KUKA KRL program: EPS_2_25694_LG03_A_20260223033042.src

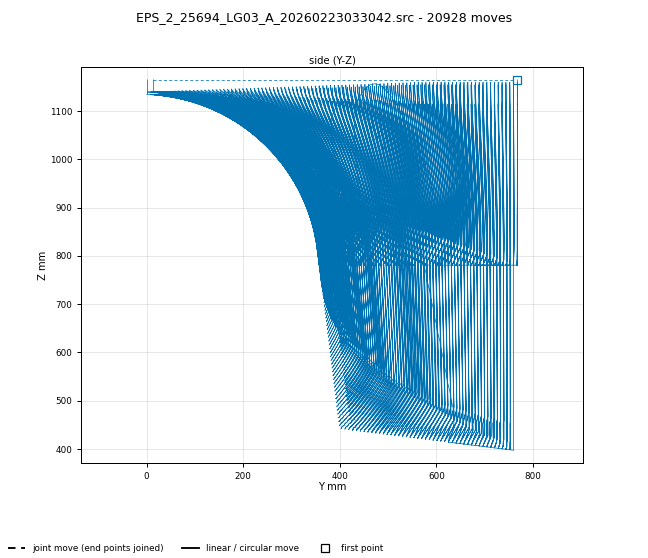
[picture p0: tool path of EPS_2_25694_LG03_A_20260223033042.src, 20928 of 20930 moves have a stored position in this frame; points joined in program order, loops and branches not executed]
&ACCESS RVP
&REL 4
&COMMENT QRS 19112012
&PARAM EDITMASK = *
DEF PART()
EXT BAS (BAS_COMMAND :IN,REAL :IN )
INT I
BAS (#INITMOV,0 )

;KUKA QRS Post kuka4.cps  Date:22-06-2017 !

File_ID=3046

QRS_PRE_INIT()

;Init var - Until changes are made in qrs_pre_init
Outlet_Square_prg=0
Inlet_1_Square_prg=0
Inlet_2_Square_prg=0
Inlet_3_Square_prg=0
Inlet_4_Square_prg=0
Inlet_5_Square_prg=0

Outlet_1={X 0.000, Y 562.000, Z 811.500, B 0.000, E1 0.000 }
Inlet_1={X 0.000, Y 562.000, Z 771.500, B 0.000, E1 183.000 }
Outlet_1_type=686
Inlet_1_type=686
;QRS#1=Sidecore dimensions
;QRS#2=675-27" Concrete
;QRS#3=675-27" Concrete
;QRS#4=
;QRS#5=
;QRS#6=
;QRS#7=
;QRS#8=
;QRS#9=S306-38L
;QRS#10=S306-38L
;QRS#11=
;QRS#12=
;QRS#13=
;QRS#14=
;QRS#15=
;QRS#16=1524x152x1600 5,25'
;QRS#17=EPS Height
;QRS#18=1154,5
;QRS#19=*
;QRS#20= UPDATED VERSION 22-06-2017
;QRS#21=*
Outlet_Square=0550
Inlet_1_Square=0550
Inlet_2_Square=0
Inlet_3_Square=0
Inlet_4_Square=0
Inlet_5_Square=0
Mill_Square=1
Outlet_Square_Prg=265
Inlet_1_Square_prg=265

QRS_INIT()

$ADVANCE=5

; T1
PTP {E1 173.017,E2 173.017}
PTP {X 0,Y 767.74,A -85,B 0,C 180,E1 173.017,E2 173.017,E3 0,E4 0,E5 0,E6 0}
QRS_SPEED_INIT()
LIN {X 0,Y 767.74,Z 1164.5,A -85,B 0,C 180,E1 173.017,E2 173.017,E3 0,E4 0,E5 0,E6 0} C_VEL
LIN {X 0,Y 767.74,Z 782.81,A -85,B 0,C 180,E1 173.017,E2 173.017} C_VEL
LIN {X 0,Y 767.776,Z 780.81,A -85,B 0,C 180,E1 173.166,E2 173.166} C_VEL
LIN {X 0,Y 767.86,Z 780.81,A -85,B 0,C 180,E1 173.458,E2 173.458} C_VEL
LIN {X 0,Y 767.876,Z 780.81,A -85,B 0,C 180,E1 177.201,E2 177.201} C_VEL
LIN {X 0,Y 767.864,Z 780.81,A -85,B 0,C 180,E1 180.933,E2 180.933} C_VEL
LIN {X 0,Y 767.829,Z 780.81,A -85,B 0,C 180,E1 184.668,E2 184.668} C_VEL
LIN {X 0,Y 767.837,Z 780.81,A -85,B 0,C 180,E1 188.423,E2 188.423} C_VEL
LIN {X 0,Y 767.822,Z 780.81,A -85,B 0,C 180,E1 192.215,E2 192.215} C_VEL
LIN {X 0,Y 767.843,Z 780.81,A -85,B 0,C 180,E1 196.207,E2 196.207} C_VEL
LIN {X 0,Y 767.794,Z 780.81,A -85,B 0,C 180,E1 199.987,E2 199.987} C_VEL
LIN {X 0,Y 767.77,Z 780.81,A -85,B 0,C 180,E1 204.012,E2 204.012} C_VEL
LIN {X 0,Y 767.76,Z 780.81,A -85,B 0,C 180,E1 208.167,E2 208.167} C_VEL
LIN {X 0,Y 767.325,Z 780.81,A -85,B 0,C 180,E1 210.324,E2 210.324} C_VEL
LIN {X 0,Y 767.754,Z 780.81,A -85,B 0,C 180,E1 212.49,E2 212.49} C_VEL
LIN {X 0,Y 767.438,Z 780.81,A -85,B 0,C 180,E1 213.851,E2 213.851} C_VEL
LIN {X 0,Y 767.747,Z 780.81,A -85,B 0,C 180,E1 217.098,E2 217.098} C_VEL
LIN {X 0,Y 767.106,Z 780.81,A -85,B 0,C 180,E1 220.032,E2 220.032} C_VEL
LIN {X 0,Y 767.543,Z 780.81,A -85,B 0,C 180,E1 221.879,E2 221.879} C_VEL
LIN {X 0,Y 767.594,Z 780.81,A -85,B 0,C 180,E1 222.892,E2 222.892} C_VEL
LIN {X 0,Y 767.642,Z 780.81,A -85,B 0,C 180,E1 227.104,E2 227.104} C_VEL
LIN {X 0,Y 767.576,Z 780.81,A -85,B 0,C 180,E1 228.123,E2 228.123} C_VEL
LIN {X 0,Y 767.128,Z 780.81,A -85,B 0,C 180,E1 230.555,E2 230.555} C_VEL
LIN {X 0,Y 767.697,Z 780.81,A -85,B 0,C 180,E1 232.964,E2 232.964} C_VEL
LIN {X 0,Y 767.564,Z 780.81,A -85,B 0,C 180,E1 236.135,E2 236.135} C_VEL
LIN {X 0,Y 767.581,Z 780.81,A -85,B 0,C 180,E1 237.502,E2 237.502} C_VEL
LIN {X 0,Y 767.865,Z 780.81,A -85,B 0,C 180,E1 240.355,E2 240.355} C_VEL
LIN {X 0,Y 766.729,Z 780.81,A -85,B 0,C 180,E1 240.572,E2 240.572} C_VEL
LIN {X 0,Y 767.117,Z 792.661,A -85,B 0,C 180,E1 240.732,E2 240.732} C_VEL
LIN {X 0,Y 767.453,Z 812.698,A -85,B 0,C 180,E1 240.956,E2 240.956} C_VEL
LIN {X 0,Y 767.54,Z 837.78,A -85,B 0,C 180,E1 241.233,E2 241.233} C_VEL
LIN {X 0,Y 767.435,Z 851.279,A -85,B 0,C 180,E1 241.406,E2 241.406} C_VEL
LIN {X 0,Y 767.547,Z 867.121,A -85,B 0,C 180,E1 241.677,E2 241.677} C_VEL
LIN {X 0,Y 767.447,Z 883.749,A -85,B 0,C 180,E1 242.019,E2 242.019} C_VEL
LIN {X 0,Y 767.661,Z 900.863,A -85,B 0,C 180,E1 242.455,E2 242.455} C_VEL
LIN {X 0,Y 767.658,Z 916.823,A -85,B 0,C 180,E1 242.921,E2 242.921} C_VEL
LIN {X 0,Y 767.551,Z 930.901,A -85,B 0,C 180,E1 243.38,E2 243.38} C_VEL
LIN {X 0,Y 767.692,Z 947.263,A -85,B 0,C 180,E1 243.998,E2 243.998} C_VEL
LIN {X 0,Y 767.654,Z 964.029,A -85,B 0,C 180,E1 244.706,E2 244.706} C_VEL
LIN {X 0,Y 767.705,Z 977.803,A -85,B 0,C 180,E1 245.351,E2 245.351} C_VEL
LIN {X 0,Y 767.711,Z 992.578,A -85,B 0,C 180,E1 246.114,E2 246.114} C_VEL
LIN {X 0,Y 767.692,Z 1006.073,A -85,B 0,C 180,E1 246.876,E2 246.876} C_VEL
LIN {X 0,Y 767.693,Z 1018.43,A -85,B 0,C 180,E1 247.634,E2 247.634} C_VEL
LIN {X 0,Y 767.706,Z 1031.659,A -85,B 0,C 180,E1 248.522,E2 248.522} C_VEL
LIN {X 0,Y 767.725,Z 1044.179,A -85,B 0,C 180,E1 249.438,E2 249.438} C_VEL
LIN {X 0,Y 767.622,Z 1056.057,A -85,B 0,C 180,E1 250.38,E2 250.38} C_VEL
LIN {X 0,Y 767.656,Z 1066.133,A -85,B 0,C 180,E1 251.245,E2 251.245} C_VEL
LIN {X 0,Y 767.776,Z 1076.684,A -85,B 0,C 180,E1 252.23,E2 252.23} C_VEL
LIN {X 0,Y 767.631,Z 1087.458,A -85,B 0,C 180,E1 253.325,E2 253.325} C_VEL
LIN {X 0,Y 767.689,Z 1096.421,A -85,B 0,C 180,E1 254.322,E2 254.322} C_VEL
LIN {X 0,Y 767.753,Z 1104.418,A -85,B 0,C 180,E1 255.29,E2 255.29} C_VEL
LIN {X 0,Y 767.609,Z 1113.841,A -85,B 0,C 180,E1 256.548,E2 256.548} C_VEL
LIN {X 0,Y 767.734,Z 1120.549,A -85,B 0,C 180,E1 257.544,E2 257.544} C_VEL
LIN {X 0,Y 767.734,Z 1124.909,A -85,B 0,C 180,E1 258.26,E2 258.26} C_VEL
LIN {X 0,Y 767.583,Z 1129.116,A -85,B 0,C 180,E1 258.971,E2 258.971} C_VEL
LIN {X 0,Y 767.572,Z 1135.348,A -85,B 0,C 180,E1 260.157,E2 260.157} C_VEL
LIN {X 0,Y 767.811,Z 1140.751,A -85,B 0,C 180,E1 261.341,E2 261.341} C_VEL
LIN {X 0,Y 767.547,Z 1145.483,A -85,B 0,C 180,E1 262.516,E2 262.516} C_VEL
LIN {X 0,Y 767.632,Z 1149.817,A -85,B 0,C 180,E1 263.832,E2 263.832} C_VEL
LIN {X 0,Y 767.823,Z 1151.823,A -85,B 0,C 180,E1 264.583,E2 264.583} C_VEL
LIN {X 0,Y 767.649,Z 1153.68,A -85,B 0,C 180,E1 265.331,E2 265.331} C_VEL
LIN {X 0,Y 767.55,Z 1155.934,A -85,B 0,C 180,E1 266.453,E2 266.453} C_VEL
LIN {X 0,Y 767.663,Z 1157.027,A -85,B 0,C 180,E1 267.201,E2 267.201} C_VEL
LIN {X 0,Y 767.835,Z 1157.84,A -85,B 0,C 180,E1 267.948,E2 267.948} C_VEL
LIN {X 0,Y 767.554,Z 1158.708,A -85,B 0,C 180,E1 269.067,E2 269.067} C_VEL
LIN {X 0,Y 767.695,Z 1158.681,A -85,B 0,C 180,E1 270.933,E2 270.933} C_VEL
LIN {X 0,Y 767.64,Z 1157.878,A -85,B 0,C 180,E1 272.053,E2 272.053} C_VEL
LIN {X 0,Y 767.509,Z 1157.056,A -85,B 0,C 180,E1 272.8,E2 272.8} C_VEL
LIN {X 0,Y 767.499,Z 1155.944,A -85,B 0,C 180,E1 273.547,E2 273.547} C_VEL
LIN {X 0,Y 767.785,Z 1152.857,A -85,B 0,C 180,E1 275.043,E2 275.043} C_VEL
LIN {X 0,Y 767.582,Z 1149.826,A -85,B 0,C 180,E1 276.169,E2 276.169} C_VEL
LIN {X 0,Y 767.707,Z 1145.456,A -85,B 0,C 180,E1 277.483,E2 277.483} C_VEL
LIN {X 0,Y 767.822,Z 1143.577,A -85,B 0,C 180,E1 277.952,E2 277.952} C_VEL
LIN {X 0,Y 767.616,Z 1139.757,A -85,B 0,C 180,E1 278.897,E2 278.897} C_VEL
LIN {X 0,Y 767.551,Z 1134.196,A -85,B 0,C 180,E1 280.08,E2 280.08} C_VEL
LIN {X 0,Y 767.824,Z 1127.78,A -85,B 0,C 180,E1 281.263,E2 281.263} C_VEL
LIN {X 0,Y 767.618,Z 1120.562,A -85,B 0,C 180,E1 282.457,E2 282.457} C_VEL
LIN {X 0,Y 767.66,Z 1112.697,A -85,B 0,C 180,E1 283.613,E2 283.613} C_VEL
LIN {X 0,Y 767.827,Z 1105.878,A -85,B 0,C 180,E1 284.516,E2 284.516} C_VEL
LIN {X 0,Y 767.632,Z 1096.425,A -85,B 0,C 180,E1 285.679,E2 285.679} C_VEL
LIN {X 0,Y 767.732,Z 1085.175,A -85,B 0,C 180,E1 286.916,E2 286.916} C_VEL
LIN {X 0,Y 767.752,Z 1075.434,A -85,B 0,C 180,E1 287.893,E2 287.893} C_VEL
LIN {X 0,Y 767.661,Z 1064.764,A -85,B 0,C 180,E1 288.878,E2 288.878} C_VEL
LIN {X 0,Y 767.747,Z 1053.06,A -85,B 0,C 180,E1 289.864,E2 289.864} C_VEL
LIN {X 0,Y 767.721,Z 1040.925,A -85,B 0,C 180,E1 290.807,E2 290.807} C_VEL
LIN {X 0,Y 767.697,Z 1029.991,A -85,B 0,C 180,E1 291.595,E2 291.595} C_VEL
LIN {X 0,Y 767.713,Z 1016.406,A -85,B 0,C 180,E1 292.491,E2 292.491} C_VEL
LIN {X 0,Y 767.708,Z 1002.8,A -85,B 0,C 180,E1 293.314,E2 293.314} C_VEL
LIN {X 0,Y 767.702,Z 989.124,A -85,B 0,C 180,E1 294.071,E2 294.071} C_VEL
LIN {X 0,Y 767.609,Z 974.312,A -85,B 0,C 180,E1 294.82,E2 294.82} C_VEL
LIN {X 0,Y 767.699,Z 960.654,A -85,B 0,C 180,E1 295.444,E2 295.444} C_VEL
LIN {X 0,Y 767.675,Z 945.45,A -85,B 0,C 180,E1 296.074,E2 296.074} C_VEL
LIN {X 0,Y 767.621,Z 931.718,A -85,B 0,C 180,E1 296.587,E2 296.587} C_VEL
LIN {X 0,Y 767.676,Z 913.476,A -85,B 0,C 180,E1 297.183,E2 297.183} C_VEL
LIN {X 0,Y 767.512,Z 896.544,A -85,B 0,C 180,E1 297.665,E2 297.665} C_VEL
LIN {X 0,Y 767.581,Z 885.096,A -85,B 0,C 180,E1 297.943,E2 297.943} C_VEL
LIN {X 0,Y 767.624,Z 871.462,A -85,B 0,C 180,E1 298.231,E2 298.231} C_VEL
LIN {X 0,Y 767.575,Z 862.13,A -85,B 0,C 180,E1 298.41,E2 298.41} C_VEL
LIN {X 0,Y 767.446,Z 851.314,A -85,B 0,C 180,E1 298.593,E2 298.593} C_VEL
LIN {X 0,Y 767.554,Z 833.082,A -85,B 0,C 180,E1 298.825,E2 298.825} C_VEL
LIN {X 0,Y 767.414,Z 805.33,A -85,B 0,C 180,E1 299.123,E2 299.123} C_VEL
LIN {X 0,Y 767.837,Z 780.81,A -85,B 0,C 180,E1 299.711,E2 299.711} C_VEL
LIN {X 0,Y 767.787,Z 780.81,A -85,B 0,C 180,E1 302.489,E2 302.489} C_VEL
LIN {X 0,Y 767.256,Z 780.81,A -85,B 0,C 180,E1 304.756,E2 304.756} C_VEL
LIN {X 0,Y 767.702,Z 780.81,A -85,B 0,C 180,E1 307.094,E2 307.094} C_VEL
LIN {X 0,Y 767.16,Z 780.81,A -85,B 0,C 180,E1 310.037,E2 310.037} C_VEL
LIN {X 0,Y 767.662,Z 780.81,A -85,B 0,C 180,E1 311.871,E2 311.871} C_VEL
LIN {X 0,Y 767.7,Z 780.81,A -85,B 0,C 180,E1 312.901,E2 312.901} C_VEL
LIN {X 0,Y 767.677,Z 780.81,A -85,B 0,C 180,E1 314.427,E2 314.427} C_VEL
LIN {X 0,Y 767.632,Z 780.81,A -85,B 0,C 180,E1 315.57,E2 315.57} C_VEL
LIN {X 0,Y 767.691,Z 780.81,A -85,B 0,C 180,E1 319.916,E2 319.916} C_VEL
LIN {X 0,Y 767.696,Z 780.81,A -85,B 0,C 180,E1 320.59,E2 320.59} C_VEL
LIN {X 0,Y 767.232,Z 780.81,A -85,B 0,C 180,E1 322.953,E2 322.953} C_VEL
LIN {X 0,Y 767.727,Z 780.81,A -85,B 0,C 180,E1 325.269,E2 325.269} C_VEL
LIN {X 0,Y 767.773,Z 780.81,A -85,B 0,C 180,E1 329.619,E2 329.619} C_VEL
LIN {X 0,Y 767.785,Z 780.81,A -85,B 0,C 180,E1 333.537,E2 333.537} C_VEL
LIN {X 0,Y 767.777,Z 780.81,A -85,B 0,C 180,E1 333.929,E2 333.929} C_VEL
LIN {X 0,Y 767.78,Z 780.81,A -85,B 0,C 180,E1 338.015,E2 338.015} C_VEL
LIN {X 0,Y 767.809,Z 780.81,A -85,B 0,C 180,E1 341.986,E2 341.986} C_VEL
LIN {X 0,Y 767.512,Z 780.81,A -85,B 0,C 180,E1 343.93,E2 343.93} C_VEL
LIN {X 0,Y 767.651,Z 780.81,A -85,B 0,C 180,E1 345.866,E2 345.866} C_VEL
LIN {X 0,Y 767.836,Z 780.81,A -85,B 0,C 180,E1 349.687,E2 349.687} C_VEL
LIN {X 0,Y 767.821,Z 780.81,A -85,B 0,C 180,E1 353.458,E2 353.458} C_VEL
LIN {X 0,Y 767.843,Z 780.81,A -85,B 0,C 180,E1 357.201,E2 357.201} C_VEL
LIN {X 0,Y 767.846,Z 780.81,A -85,B 0,C 180,E1 360.933,E2 360.933} C_VEL
LIN {X 0,Y 767.867,Z 780.81,A -85,B 0,C 180,E1 364.668,E2 364.668} C_VEL
LIN {X 0,Y 767.85,Z 780.81,A -85,B 0,C 180,E1 368.423,E2 368.423} C_VEL
LIN {X 0,Y 767.826,Z 780.81,A -85,B 0,C 180,E1 372.215,E2 372.215} C_VEL
LIN {X 0,Y 767.846,Z 780.81,A -85,B 0,C 180,E1 376.208,E2 376.208} C_VEL
LIN {X 0,Y 767.763,Z 780.81,A -85,B 0,C 180,E1 379.988,E2 379.988} C_VEL
LIN {X 0,Y 767.743,Z 780.81,A -85,B 0,C 180,E1 384.013,E2 384.013} C_VEL
LIN {X 0,Y 767.738,Z 780.81,A -85,B 0,C 180,E1 388.168,E2 388.168} C_VEL
LIN {X 0,Y 767.325,Z 780.81,A -85,B 0,C 180,E1 390.324,E2 390.324} C_VEL
LIN {X 0,Y 767.75,Z 780.81,A -85,B 0,C 180,E1 392.49,E2 392.49} C_VEL
LIN {X 0,Y 767.422,Z 780.81,A -85,B 0,C 180,E1 393.849,E2 393.849} C_VEL
LIN {X 0,Y 767.691,Z 780.81,A -85,B 0,C 180,E1 397.093,E2 397.093} C_VEL
LIN {X 0,Y 767.108,Z 780.81,A -85,B 0,C 180,E1 400.032,E2 400.032} C_VEL
LIN {X 0,Y 767.596,Z 780.81,A -85,B 0,C 180,E1 401.875,E2 401.875} C_VEL
LIN {X 0,Y 767.635,Z 780.81,A -85,B 0,C 180,E1 402.895,E2 402.895} C_VEL
LIN {X 0,Y 767.63,Z 780.81,A -85,B 0,C 180,E1 404.43,E2 404.43} C_VEL
LIN {X 0,Y 767.609,Z 780.81,A -85,B 0,C 180,E1 405.568,E2 405.568} C_VEL
LIN {X 0,Y 767.614,Z 780.81,A -85,B 0,C 180,E1 409.923,E2 409.923} C_VEL
LIN {X 0,Y 767.676,Z 780.81,A -85,B 0,C 180,E1 410.589,E2 410.589} C_VEL
LIN {X 0,Y 767.696,Z 780.81,A -85,B 0,C 180,E1 412.964,E2 412.964} C_VEL
LIN {X 0,Y 767.339,Z 780.81,A -85,B 0,C 180,E1 415.248,E2 415.248} C_VEL
LIN {X 0,Y 767.821,Z 780.81,A -85,B 0,C 180,E1 417.836,E2 417.836} C_VEL
LIN {X 0,Y 767.17,Z 780.81,A -85,B 0,C 180,E1 417.966,E2 417.966} C_VEL
LIN {X 0,Y 767.625,Z 808.807,A -85,B 0,C 180,E1 418.329,E2 418.329} C_VEL
LIN {X 0,Y 767.563,Z 827.01,A -85,B 0,C 180,E1 418.63,E2 418.63} C_VEL
LIN {X 0,Y 767.462,Z 835.654,A -85,B 0,C 180,E1 418.803,E2 418.803} C_VEL
LIN {X 0,Y 767.61,Z 845.009,A -85,B 0,C 180,E1 419.011,E2 419.011} C_VEL
LIN {X 0,Y 767.634,Z 860.435,A -85,B 0,C 180,E1 419.397,E2 419.397} C_VEL
LIN {X 0,Y 767.509,Z 876.238,A -85,B 0,C 180,E1 419.851,E2 419.851} C_VEL
LIN {X 0,Y 767.671,Z 892.53,A -85,B 0,C 180,E1 420.4,E2 420.4} C_VEL
LIN {X 0,Y 767.68,Z 908.704,A -85,B 0,C 180,E1 421.012,E2 421.012} C_VEL
LIN {X 0,Y 767.654,Z 922.098,A -85,B 0,C 180,E1 421.571,E2 421.571} C_VEL
LIN {X 0,Y 767.712,Z 937.549,A -85,B 0,C 180,E1 422.293,E2 422.293} C_VEL
LIN {X 0,Y 767.705,Z 952.053,A -85,B 0,C 180,E1 423.039,E2 423.039} C_VEL
LIN {X 0,Y 767.71,Z 965.906,A -85,B 0,C 180,E1 423.821,E2 423.821} C_VEL
LIN {X 0,Y 767.717,Z 980.172,A -85,B 0,C 180,E1 424.706,E2 424.706} C_VEL
LIN {X 0,Y 767.75,Z 991.735,A -85,B 0,C 180,E1 425.484,E2 425.484} C_VEL
LIN {X 0,Y 767.674,Z 1003.871,A -85,B 0,C 180,E1 426.367,E2 426.367} C_VEL
LIN {X 0,Y 767.673,Z 1015.104,A -85,B 0,C 180,E1 427.255,E2 427.255} C_VEL
LIN {X 0,Y 767.763,Z 1027.004,A -85,B 0,C 180,E1 428.283,E2 428.283} C_VEL
LIN {X 0,Y 767.656,Z 1036.937,A -85,B 0,C 180,E1 429.208,E2 429.208} C_VEL
LIN {X 0,Y 767.716,Z 1047.241,A -85,B 0,C 180,E1 430.259,E2 430.259} C_VEL
LIN {X 0,Y 767.763,Z 1055.099,A -85,B 0,C 180,E1 431.125,E2 431.125} C_VEL
LIN {X 0,Y 767.611,Z 1064.298,A -85,B 0,C 180,E1 432.226,E2 432.226} C_VEL
LIN {X 0,Y 767.757,Z 1073.448,A -85,B 0,C 180,E1 433.45,E2 433.45} C_VEL
LIN {X 0,Y 767.761,Z 1078.038,A -85,B 0,C 180,E1 434.13,E2 434.13} C_VEL
LIN {X 0,Y 767.637,Z 1081.873,A -85,B 0,C 180,E1 434.708,E2 434.708} C_VEL
LIN {X 0,Y 767.604,Z 1088.786,A -85,B 0,C 180,E1 435.865,E2 435.865} C_VEL
LIN {X 0,Y 767.792,Z 1095.097,A -85,B 0,C 180,E1 437.067,E2 437.067} C_VEL
LIN {X 0,Y 767.589,Z 1100.644,A -85,B 0,C 180,E1 438.258,E2 438.258} C_VEL
LIN {X 0,Y 767.643,Z 1104.446,A -85,B 0,C 180,E1 439.21,E2 439.21} C_VEL
LIN {X 0,Y 767.824,Z 1107.736,A -85,B 0,C 180,E1 440.16,E2 440.16} C_VEL
LIN {X 0,Y 767.702,Z 1109.353,A -85,B 0,C 180,E1 440.631,E2 440.631} C_VEL
LIN {X 0,Y 767.567,Z 1113.194,A -85,B 0,C 180,E1 442.045,E2 442.045} C_VEL
LIN {X 0,Y 767.789,Z 1115.494,A -85,B 0,C 180,E1 443.158,E2 443.158} C_VEL
LIN {X 0,Y 767.831,Z 1115.954,A -85,B 0,C 180,E1 443.458,E2 443.458} C_VEL
LIN {X 0,Y 767.624,Z 1117.112,A -85,B 0,C 180,E1 444.207,E2 444.207} C_VEL
LIN {X 0,Y 767.512,Z 1118.283,A -85,B 0,C 180,E1 445.33,E2 445.33} C_VEL
LIN {X 0,Y 767.698,Z 1118.806,A -85,B 0,C 180,E1 446.453,E2 446.453} C_VEL
LIN {X 0,Y 767.748,Z 1118.875,A -85,B 0,C 180,E1 447.201,E2 447.201} C_VEL
LIN {X 0,Y 767.507,Z 1117.851,A -85,B 0,C 180,E1 449.067,E2 449.067} C_VEL
LIN {X 0,Y 767.644,Z 1116.942,A -85,B 0,C 180,E1 449.813,E2 449.813} C_VEL
LIN {X 0,Y 767.711,Z 1115.125,A -85,B 0,C 180,E1 450.933,E2 450.933} C_VEL
LIN {X 0,Y 767.545,Z 1112.754,A -85,B 0,C 180,E1 452.053,E2 452.053} C_VEL
LIN {X 0,Y 767.684,Z 1109.673,A -85,B 0,C 180,E1 453.173,E2 453.173} C_VEL
LIN {X 0,Y 767.786,Z 1107.173,A -85,B 0,C 180,E1 453.92,E2 453.92} C_VEL
LIN {X 0,Y 767.599,Z 1104.58,A -85,B 0,C 180,E1 454.669,E2 454.669} C_VEL
LIN {X 0,Y 767.553,Z 1100.045,A -85,B 0,C 180,E1 455.794,E2 455.794} C_VEL
LIN {X 0,Y 767.785,Z 1094.666,A -85,B 0,C 180,E1 456.935,E2 456.935} C_VEL
LIN {X 0,Y 767.596,Z 1087.996,A -85,B 0,C 180,E1 458.19,E2 458.19} C_VEL
LIN {X 0,Y 767.652,Z 1080.845,A -85,B 0,C 180,E1 459.369,E2 459.369} C_VEL
LIN {X 0,Y 767.791,Z 1074.425,A -85,B 0,C 180,E1 460.314,E2 460.314} C_VEL
LIN {X 0,Y 767.664,Z 1069.239,A -85,B 0,C 180,E1 461.028,E2 461.028} C_VEL
LIN {X 0,Y 767.628,Z 1063.812,A -85,B 0,C 180,E1 461.742,E2 461.742} C_VEL
LIN {X 0,Y 767.784,Z 1054.842,A -85,B 0,C 180,E1 462.813,E2 462.813} C_VEL
LIN {X 0,Y 767.664,Z 1044.529,A -85,B 0,C 180,E1 463.937,E2 463.937} C_VEL
LIN {X 0,Y 767.652,Z 1034.84,A -85,B 0,C 180,E1 464.905,E2 464.905} C_VEL
LIN {X 0,Y 767.78,Z 1024.295,A -85,B 0,C 180,E1 465.87,E2 465.87} C_VEL
LIN {X 0,Y 767.69,Z 1013.391,A -85,B 0,C 180,E1 466.795,E2 466.795} C_VEL
LIN {X 0,Y 767.661,Z 1000.796,A -85,B 0,C 180,E1 467.773,E2 467.773} C_VEL
LIN {X 0,Y 767.698,Z 988.777,A -85,B 0,C 180,E1 468.631,E2 468.631} C_VEL
LIN {X 0,Y 767.696,Z 975.626,A -85,B 0,C 180,E1 469.494,E2 469.494} C_VEL
LIN {X 0,Y 767.704,Z 962.607,A -85,B 0,C 180,E1 470.28,E2 470.28} C_VEL
LIN {X 0,Y 767.697,Z 948.636,A -85,B 0,C 180,E1 471.051,E2 471.051} C_VEL
LIN {X 0,Y 767.707,Z 934.96,A -85,B 0,C 180,E1 471.742,E2 471.742} C_VEL
LIN {X 0,Y 767.647,Z 919.959,A -85,B 0,C 180,E1 472.43,E2 472.43} C_VEL
LIN {X 0,Y 767.694,Z 904.586,A -85,B 0,C 180,E1 473.061,E2 473.061} C_VEL
LIN {X 0,Y 767.65,Z 889.027,A -85,B 0,C 180,E1 473.634,E2 473.634} C_VEL
LIN {X 0,Y 767.507,Z 874.368,A -85,B 0,C 180,E1 474.119,E2 474.119} C_VEL
LIN {X 0,Y 767.638,Z 856.271,A -85,B 0,C 180,E1 474.622,E2 474.622} C_VEL
LIN {X 0,Y 767.519,Z 839.771,A -85,B 0,C 180,E1 475.021,E2 475.021} C_VEL
LIN {X 0,Y 767.506,Z 831.89,A -85,B 0,C 180,E1 475.182,E2 475.182} C_VEL
LIN {X 0,Y 767.611,Z 825.775,A -85,B 0,C 180,E1 475.303,E2 475.303} C_VEL
LIN {X 0,Y 767.642,Z 810.141,A -85,B 0,C 180,E1 475.559,E2 475.559} C_VEL
LIN {X 0,Y 767.332,Z 792.046,A -85,B 0,C 180,E1 475.801,E2 475.801} C_VEL
LIN {X 0,Y 766.199,Z 783.819,A -85,B 0,C 180,E1 475.934,E2 475.934} C_VEL
LIN {X 0,Y 765.808,Z 780.81,A -85,B 0,C 180,E1 475.999,E2 475.999} C_VEL
LIN {X 0,Y 767.122,Z 780.81,A -85,B 0,C 180,E1 476.095,E2 476.095} C_VEL
LIN {X 0,Y 767.838,Z 780.81,A -85,B 0,C 180,E1 476.471,E2 476.471} C_VEL
LIN {X 0,Y 767.806,Z 780.81,A -85,B 0,C 180,E1 478.165,E2 478.165} C_VEL
LIN {X 0,Y 767.75,Z 780.81,A -85,B 0,C 180,E1 482.49,E2 482.49} C_VEL
LIN {X 0,Y 767.423,Z 780.81,A -85,B 0,C 180,E1 483.849,E2 483.849} C_VEL
LIN {X 0,Y 767.68,Z 780.81,A -85,B 0,C 180,E1 487.092,E2 487.092} C_VEL
LIN {X 0,Y 767.11,Z 780.81,A -85,B 0,C 180,E1 490.032,E2 490.032} C_VEL
LIN {X 0,Y 767.605,Z 780.81,A -85,B 0,C 180,E1 491.875,E2 491.875} C_VEL
LIN {X 0,Y 767.631,Z 780.81,A -85,B 0,C 180,E1 492.895,E2 492.895} C_VEL
LIN {X 0,Y 767.632,Z 780.81,A -85,B 0,C 180,E1 494.43,E2 494.43} C_VEL
LIN {X 0,Y 767.608,Z 780.81,A -85,B 0,C 180,E1 495.568,E2 495.568} C_VEL
LIN {X 0,Y 767.62,Z 780.81,A -85,B 0,C 180,E1 499.922,E2 499.922} C_VEL
LIN {X 0,Y 767.606,Z 780.81,A -85,B 0,C 180,E1 500.584,E2 500.584} C_VEL
LIN {X 0,Y 767.183,Z 780.81,A -85,B 0,C 180,E1 502.957,E2 502.957} C_VEL
LIN {X 0,Y 767.715,Z 780.81,A -85,B 0,C 180,E1 505.268,E2 505.268} C_VEL
LIN {X 0,Y 767.763,Z 780.81,A -85,B 0,C 180,E1 509.621,E2 509.621} C_VEL
LIN {X 0,Y 767.767,Z 780.81,A -85,B 0,C 180,E1 513.54,E2 513.54} C_VEL
LIN {X 0,Y 767.758,Z 780.81,A -85,B 0,C 180,E1 513.929,E2 513.929} C_VEL
LIN {X 0,Y 767.768,Z 780.81,A -85,B 0,C 180,E1 518.014,E2 518.014} C_VEL
LIN {X 0,Y 767.802,Z 780.81,A -85,B 0,C 180,E1 521.986,E2 521.986} C_VEL
LIN {X 0,Y 767.532,Z 780.81,A -85,B 0,C 180,E1 523.931,E2 523.931} C_VEL
LIN {X 0,Y 767.66,Z 780.81,A -85,B 0,C 180,E1 525.866,E2 525.866} C_VEL
LIN {X 0,Y 767.851,Z 780.81,A -85,B 0,C 180,E1 529.687,E2 529.687} C_VEL
LIN {X 0,Y 767.776,Z 780.81,A -85,B 0,C 180,E1 533.166,E2 533.166} C_VEL
LIN {X 0,Y 765.242,Z 780.81,A -85,B 0,C 180,E1 534.125,E2 534.125} C_VEL
LIN {X 0,Y 759.665,Z 780.81,A -85,B 0,C 180,E1 535.553,E2 535.553} C_VEL
LIN {X 0,Y 759.584,Z 780.81,A -85,B 0,C 180,E1 535.719,E2 535.719} C_VEL
LIN {X 0,Y 759.687,Z 780.81,A -85,B 0,C 180,E1 539.998,E2 539.998} C_VEL
LIN {X 0,Y 759.881,Z 780.81,A -85,B 0,C 180,E1 544.56,E2 544.56} C_VEL
LIN {X 0,Y 759.686,Z 780.81,A -85,B 0,C 180,E1 549.153,E2 549.153} C_VEL
LIN {X 0,Y 759.484,Z 780.81,A -85,B 0,C 180,E1 553.809,E2 553.809} C_VEL
LIN {X 0,Y 759.583,Z 780.81,A -85,B 0,C 180,E1 557.357,E2 557.357} C_VEL
LIN {X 0,Y 759.55,Z 780.81,A -85,B 0,C 180,E1 560.978,E2 560.978} C_VEL
LIN {X 0,Y 759.605,Z 780.81,A -85,B 0,C 180,E1 564.687,E2 564.687} C_VEL
LIN {X 0,Y 759.603,Z 780.81,A -85,B 0,C 180,E1 568.917,E2 568.917} C_VEL
LIN {X 0,Y 759.635,Z 780.81,A -85,B 0,C 180,E1 573.332,E2 573.332} C_VEL
LIN {X 0,Y 759.426,Z 780.81,A -85,B 0,C 180,E1 578.076,E2 578.076} C_VEL
LIN {X 0,Y 759.685,Z 780.81,A -85,B 0,C 180,E1 582.609,E2 582.609} C_VEL
LIN {X 0,Y 759.713,Z 780.81,A -85,B 0,C 180,E1 587.446,E2 587.446} C_VEL
LIN {X 0,Y 759.656,Z 780.81,A -85,B 0,C 180,E1 593.361,E2 593.361} C_VEL
LIN {X 0,Y 759.694,Z 780.81,A -85,B 0,C 180,E1 597.516,E2 597.516} C_VEL
LIN {X 0,Y 759.71,Z 781.308,A -85,B 0,C 180,E1 600.297,E2 600.297} C_VEL
LIN {X 0,Y 760.544,Z 861.196,A -85,B 0,C 180,E1 601.287,E2 601.287} C_VEL
LIN {X 0,Y 760.585,Z 901.893,A -85,B 0,C 180,E1 602.207,E2 602.207} C_VEL
LIN {X 0,Y 760.439,Z 944.766,A -85,B 0,C 180,E1 603.633,E2 603.633} C_VEL
LIN {X 0,Y 760.322,Z 985.63,A -85,B 0,C 180,E1 605.5,E2 605.5} C_VEL
LIN {X 0,Y 760.131,Z 1022.191,A -85,B 0,C 180,E1 607.653,E2 607.653} C_VEL
LIN {X 0,Y 759.965,Z 1056.853,A -85,B 0,C 180,E1 610.243,E2 610.243} C_VEL
LIN {X 0,Y 759.869,Z 1086.946,A -85,B 0,C 180,E1 613.091,E2 613.091} C_VEL
LIN {X 0,Y 759.801,Z 1112.414,A -85,B 0,C 180,E1 616.192,E2 616.192} C_VEL
LIN {X 0,Y 759.703,Z 1130.679,A -85,B 0,C 180,E1 619.107,E2 619.107} C_VEL
LIN {X 0,Y 759.715,Z 1145.249,A -85,B 0,C 180,E1 622.283,E2 622.283} C_VEL
LIN {X 0,Y 759.768,Z 1154.484,A -85,B 0,C 180,E1 625.436,E2 625.436} C_VEL
LIN {X 0,Y 759.709,Z 1159.172,A -85,B 0,C 180,E1 628.86,E2 628.86} C_VEL
LIN {X 0,Y 759.722,Z 1158.226,A -85,B 0,C 180,E1 632.279,E2 632.279} C_VEL
LIN {X 0,Y 759.753,Z 1151.677,A -85,B 0,C 180,E1 635.707,E2 635.707} C_VEL
LIN {X 0,Y 759.777,Z 1140.638,A -85,B 0,C 180,E1 638.866,E2 638.866} C_VEL
LIN {X 0,Y 759.807,Z 1123.983,A -85,B 0,C 180,E1 642.053,E2 642.053} C_VEL
LIN {X 0,Y 759.907,Z 1102.324,A -85,B 0,C 180,E1 645.128,E2 645.128} C_VEL
LIN {X 0,Y 759.991,Z 1075.253,A -85,B 0,C 180,E1 648.099,E2 648.099} C_VEL
LIN {X 0,Y 760.104,Z 1041.716,A -85,B 0,C 180,E1 650.967,E2 650.967} C_VEL
LIN {X 0,Y 760.244,Z 1003.273,A -85,B 0,C 180,E1 653.53,E2 653.53} C_VEL
LIN {X 0,Y 760.391,Z 962.85,A -85,B 0,C 180,E1 655.609,E2 655.609} C_VEL
LIN {X 0,Y 760.524,Z 920.491,A -85,B 0,C 180,E1 657.232,E2 657.232} C_VEL
LIN {X 0,Y 760.628,Z 881.194,A -85,B 0,C 180,E1 658.314,E2 658.314} C_VEL
LIN {X 0,Y 760.616,Z 835.869,A -85,B 0,C 180,E1 659.078,E2 659.078} C_VEL
LIN {X 0,Y 759.953,Z 780.81,A -85,B 0,C 180,E1 659.744,E2 659.744} C_VEL
LIN {X 0,Y 759.453,Z 780.81,A -85,B 0,C 180,E1 663.856,E2 663.856} C_VEL
LIN {X 0,Y 759.408,Z 780.81,A -85,B 0,C 180,E1 668.086,E2 668.086} C_VEL
LIN {X 0,Y 759.791,Z 780.81,A -85,B 0,C 180,E1 672.632,E2 672.632} C_VEL
LIN {X 0,Y 759.598,Z 780.81,A -85,B 0,C 180,E1 675.883,E2 675.883} C_VEL
LIN {X 0,Y 759.69,Z 780.81,A -85,B 0,C 180,E1 680.872,E2 680.872} C_VEL
LIN {X 0,Y 759.484,Z 780.81,A -85,B 0,C 180,E1 686.153,E2 686.153} C_VEL
LIN {X 0,Y 759.467,Z 780.81,A -85,B 0,C 180,E1 691.098,E2 691.098} C_VEL
LIN {X 0,Y 759.814,Z 780.81,A -85,B 0,C 180,E1 694.06,E2 694.06} C_VEL
LIN {X 0,Y 759.559,Z 780.81,A -85,B 0,C 180,E1 699.022,E2 699.022} C_VEL
LIN {X 0,Y 759.607,Z 780.81,A -85,B 0,C 180,E1 703.834,E2 703.834} C_VEL
LIN {X 0,Y 759.523,Z 780.81,A -85,B 0,C 180,E1 708.528,E2 708.528} C_VEL
LIN {X 0,Y 759.548,Z 780.81,A -85,B 0,C 180,E1 711.998,E2 711.998} C_VEL
LIN {X 0,Y 759.737,Z 780.81,A -85,B 0,C 180,E1 716.581,E2 716.581} C_VEL
LIN {X 0,Y 759.863,Z 780.81,A -85,B 0,C 180,E1 721.141,E2 721.141} C_VEL
LIN {X 0,Y 759.632,Z 780.81,A -85,B 0,C 180,E1 725.709,E2 725.709} C_VEL
LIN {X 0,Y 759.687,Z 780.81,A -85,B 0,C 180,E1 729.157,E2 729.157} C_VEL
LIN {X 0,Y 759.512,Z 780.81,A -85,B 0,C 180,E1 733.812,E2 733.812} C_VEL
LIN {X 0,Y 759.574,Z 780.81,A -85,B 0,C 180,E1 737.361,E2 737.361} C_VEL
LIN {X 0,Y 759.534,Z 780.81,A -85,B 0,C 180,E1 740.982,E2 740.982} C_VEL
LIN {X 0,Y 759.577,Z 780.81,A -85,B 0,C 180,E1 744.692,E2 744.692} C_VEL
LIN {X 0,Y 759.451,Z 780.81,A -85,B 0,C 180,E1 749.827,E2 749.827} C_VEL
LIN {X 0,Y 759.521,Z 780.81,A -85,B 0,C 180,E1 753.849,E2 753.849} C_VEL
LIN {X 0,Y 759.392,Z 780.81,A -85,B 0,C 180,E1 758.082,E2 758.082} C_VEL
LIN {X 0,Y 759.702,Z 780.81,A -85,B 0,C 180,E1 762.613,E2 762.613} C_VEL
LIN {X 0,Y 759.577,Z 780.81,A -85,B 0,C 180,E1 765.871,E2 765.871} C_VEL
LIN {X 0,Y 759.73,Z 780.81,A -85,B 0,C 180,E1 770.86,E2 770.86} C_VEL
LIN {X 0,Y 759.428,Z 780.81,A -85,B 0,C 180,E1 774.758,E2 774.758} C_VEL
LIN {X 0,Y 759.851,Z 780.81,A -85,B 0,C 180,E1 777.663,E2 777.663} C_VEL
LIN {X 0,Y 760.526,Z 831.542,A -85,B 0,C 180,E1 778.438,E2 778.438} C_VEL
LIN {X 0,Y 760.382,Z 876.79,A -85,B 0,C 180,E1 779.594,E2 779.594} C_VEL
LIN {X 0,Y 760.373,Z 921.364,A -85,B 0,C 180,E1 781.278,E2 781.278} C_VEL
LIN {X 0,Y 760.264,Z 964.328,A -85,B 0,C 180,E1 783.485,E2 783.485} C_VEL
LIN {X 0,Y 760.075,Z 1003.476,A -85,B 0,C 180,E1 786.12,E2 786.12} C_VEL
LIN {X 0,Y 759.924,Z 1037.005,A -85,B 0,C 180,E1 789.028,E2 789.028} C_VEL
LIN {X 0,Y 759.813,Z 1064.146,A -85,B 0,C 180,E1 792.046,E2 792.046} C_VEL
LIN {X 0,Y 759.757,Z 1084.67,A -85,B 0,C 180,E1 795.016,E2 795.016} C_VEL
LIN {X 0,Y 759.728,Z 1101.253,A -85,B 0,C 180,E1 798.237,E2 798.237} C_VEL
LIN {X 0,Y 759.698,Z 1112.148,A -85,B 0,C 180,E1 801.421,E2 801.421} C_VEL
LIN {X 0,Y 759.727,Z 1117.794,A -85,B 0,C 180,E1 804.293,E2 804.293} C_VEL
LIN {X 0,Y 759.743,Z 1119.282,A -85,B 0,C 180,E1 807.721,E2 807.721} C_VEL
LIN {X 0,Y 759.788,Z 1115.277,A -85,B 0,C 180,E1 811.14,E2 811.14} C_VEL
LIN {X 0,Y 759.768,Z 1105.676,A -85,B 0,C 180,E1 814.564,E2 814.564} C_VEL
LIN {X 0,Y 759.753,Z 1089.848,A -85,B 0,C 180,E1 818.004,E2 818.004} C_VEL
LIN {X 0,Y 759.837,Z 1070.374,A -85,B 0,C 180,E1 821.036,E2 821.036} C_VEL
LIN {X 0,Y 759.905,Z 1046.132,A -85,B 0,C 180,E1 823.953,E2 823.953} C_VEL
LIN {X 0,Y 760.032,Z 1014.597,A -85,B 0,C 180,E1 826.905,E2 826.905} C_VEL
LIN {X 0,Y 760.181,Z 977.717,A -85,B 0,C 180,E1 829.6,E2 829.6} C_VEL
LIN {X 0,Y 760.364,Z 937.41,A -85,B 0,C 180,E1 831.878,E2 831.878} C_VEL
LIN {X 0,Y 760.48,Z 895.32,A -85,B 0,C 180,E1 833.676,E2 833.676} C_VEL
LIN {X 0,Y 760.592,Z 854.934,A -85,B 0,C 180,E1 834.934,E2 834.934} C_VEL
LIN {X 0,Y 760.685,Z 810.665,A -85,B 0,C 180,E1 835.836,E2 835.836} C_VEL
LIN {X 0,Y 759.206,Z 784.434,A -85,B 0,C 180,E1 836.221,E2 836.221} C_VEL
LIN {X 0,Y 759.055,Z 780.81,A -85,B 0,C 180,E1 836.303,E2 836.303} C_VEL
LIN {X 0,Y 759.859,Z 780.81,A -85,B 0,C 180,E1 837.22,E2 837.22} C_VEL
LIN {X 0,Y 759.622,Z 780.81,A -85,B 0,C 180,E1 843.344,E2 843.344} C_VEL
LIN {X 0,Y 759.383,Z 780.81,A -85,B 0,C 180,E1 848.089,E2 848.089} C_VEL
LIN {X 0,Y 759.73,Z 780.81,A -85,B 0,C 180,E1 852.622,E2 852.622} C_VEL
LIN {X 0,Y 759.567,Z 780.81,A -85,B 0,C 180,E1 855.876,E2 855.876} C_VEL
LIN {X 0,Y 759.609,Z 780.81,A -85,B 0,C 180,E1 860.882,E2 860.882} C_VEL
LIN {X 0,Y 759.483,Z 780.81,A -85,B 0,C 180,E1 866.149,E2 866.149} C_VEL
LIN {X 0,Y 759.463,Z 780.81,A -85,B 0,C 180,E1 871.102,E2 871.102} C_VEL
LIN {X 0,Y 759.818,Z 780.81,A -85,B 0,C 180,E1 874.056,E2 874.056} C_VEL
LIN {X 0,Y 759.551,Z 780.81,A -85,B 0,C 180,E1 879.018,E2 879.018} C_VEL
LIN {X 0,Y 759.636,Z 780.81,A -85,B 0,C 180,E1 883.831,E2 883.831} C_VEL
LIN {X 0,Y 759.556,Z 780.81,A -85,B 0,C 180,E1 888.525,E2 888.525} C_VEL
LIN {X 0,Y 759.604,Z 780.81,A -85,B 0,C 180,E1 891.995,E2 891.995} C_VEL
LIN {X 0,Y 759.584,Z 780.81,A -85,B 0,C 180,E1 895.719,E2 895.719} C_VEL
LIN {X 0,Y 758.406,Z 780.81,A -85,B 0,C 180,E1 896.371,E2 896.371} C_VEL
LIN {X 0,Y 751.856,Z 780.81,A -85,B 0,C 180,E1 898.141,E2 898.141} C_VEL
LIN {X 0,Y 751.74,Z 780.81,A -85,B 0,C 180,E1 898.308,E2 898.308} C_VEL
LIN {X 0,Y 751.696,Z 780.81,A -85,B 0,C 180,E1 902.302,E2 902.302} C_VEL
LIN {X 0,Y 751.723,Z 780.81,A -85,B 0,C 180,E1 905.766,E2 905.766} C_VEL
LIN {X 0,Y 751.644,Z 780.81,A -85,B 0,C 180,E1 909.901,E2 909.901} C_VEL
LIN {X 0,Y 751.578,Z 780.81,A -85,B 0,C 180,E1 913.957,E2 913.957} C_VEL
LIN {X 0,Y 751.654,Z 780.81,A -85,B 0,C 180,E1 917.546,E2 917.546} C_VEL
LIN {X 0,Y 751.603,Z 780.81,A -85,B 0,C 180,E1 921.211,E2 921.211} C_VEL
LIN {X 0,Y 751.601,Z 780.81,A -85,B 0,C 180,E1 925.211,E2 925.211} C_VEL
LIN {X 0,Y 751.724,Z 780.81,A -85,B 0,C 180,E1 928.838,E2 928.838} C_VEL
LIN {X 0,Y 751.857,Z 780.81,A -85,B 0,C 180,E1 932.856,E2 932.856} C_VEL
LIN {X 0,Y 751.811,Z 780.81,A -85,B 0,C 180,E1 937.074,E2 937.074} C_VEL
LIN {X 0,Y 751.604,Z 780.81,A -85,B 0,C 180,E1 943.112,E2 943.112} C_VEL
LIN {X 0,Y 751.533,Z 780.81,A -85,B 0,C 180,E1 948.43,E2 948.43} C_VEL
LIN {X 0,Y 751.712,Z 780.81,A -85,B 0,C 180,E1 953.506,E2 953.506} C_VEL
LIN {X 0,Y 751.694,Z 780.81,A -85,B 0,C 180,E1 958.488,E2 958.488} C_VEL
LIN {X 0,Y 751.985,Z 781.452,A -85,B 0,C 180,E1 959.962,E2 959.962} C_VEL
LIN {X 0,Y 753.453,Z 799.004,A -85,B 0,C 180,E1 960.216,E2 960.216} C_VEL
LIN {X 0,Y 753.614,Z 863.925,A -85,B 0,C 180,E1 961.044,E2 961.044} C_VEL
LIN {X 0,Y 753.496,Z 904.485,A -85,B 0,C 180,E1 961.998,E2 961.998} C_VEL
LIN {X 0,Y 753.242,Z 946.529,A -85,B 0,C 180,E1 963.429,E2 963.429} C_VEL
LIN {X 0,Y 752.939,Z 989.654,A -85,B 0,C 180,E1 965.453,E2 965.453} C_VEL
LIN {X 0,Y 752.603,Z 1029.035,A -85,B 0,C 180,E1 967.884,E2 967.884} C_VEL
LIN {X 0,Y 752.252,Z 1063.771,A -85,B 0,C 180,E1 970.634,E2 970.634} C_VEL
LIN {X 0,Y 752.069,Z 1092.37,A -85,B 0,C 180,E1 973.52,E2 973.52} C_VEL
LIN {X 0,Y 751.931,Z 1115.194,A -85,B 0,C 180,E1 976.448,E2 976.448} C_VEL
LIN {X 0,Y 751.821,Z 1133.762,A -85,B 0,C 180,E1 979.578,E2 979.578} C_VEL
LIN {X 0,Y 751.83,Z 1146.298,A -85,B 0,C 180,E1 982.493,E2 982.493} C_VEL
LIN {X 0,Y 751.875,Z 1154.484,A -85,B 0,C 180,E1 985.388,E2 985.388} C_VEL
LIN {X 0,Y 751.81,Z 1159.172,A -85,B 0,C 180,E1 988.848,E2 988.848} C_VEL
LIN {X 0,Y 751.817,Z 1158.226,A -85,B 0,C 180,E1 992.303,E2 992.303} C_VEL
LIN {X 0,Y 751.854,Z 1151.678,A -85,B 0,C 180,E1 995.767,E2 995.767} C_VEL
LIN {X 0,Y 751.875,Z 1140.638,A -85,B 0,C 180,E1 998.96,E2 998.96} C_VEL
LIN {X 0,Y 751.949,Z 1123.984,A -85,B 0,C 180,E1 1002.181,E2 1002.181} C_VEL
LIN {X 0,Y 752.089,Z 1103.538,A -85,B 0,C 180,E1 1005.14,E2 1005.14} C_VEL
LIN {X 0,Y 752.26,Z 1075.246,A -85,B 0,C 180,E1 1008.292,E2 1008.292} C_VEL
LIN {X 0,Y 752.505,Z 1041.717,A -85,B 0,C 180,E1 1011.189,E2 1011.189} C_VEL
LIN {X 0,Y 752.82,Z 1003.619,A -85,B 0,C 180,E1 1013.757,E2 1013.757} C_VEL
LIN {X 0,Y 753.128,Z 962.031,A -85,B 0,C 180,E1 1015.912,E2 1015.912} C_VEL
LIN {X 0,Y 753.44,Z 918.707,A -85,B 0,C 180,E1 1017.57,E2 1017.57} C_VEL
LIN {X 0,Y 753.651,Z 878.763,A -85,B 0,C 180,E1 1018.651,E2 1018.651} C_VEL
LIN {X 0,Y 753.715,Z 835.869,A -85,B 0,C 180,E1 1019.37,E2 1019.37} C_VEL
LIN {X 0,Y 752.422,Z 783.412,A -85,B 0,C 180,E1 1019.997,E2 1019.997} C_VEL
LIN {X 0,Y 751.953,Z 780.81,A -85,B 0,C 180,E1 1020.071,E2 1020.071} C_VEL
LIN {X 0,Y 751.827,Z 780.81,A -85,B 0,C 180,E1 1022.865,E2 1022.865} C_VEL
LIN {X 0,Y 751.772,Z 780.81,A -85,B 0,C 180,E1 1027.085,E2 1027.085} C_VEL
LIN {X 0,Y 751.839,Z 780.81,A -85,B 0,C 180,E1 1033.106,E2 1033.106} C_VEL
LIN {X 0,Y 751.404,Z 780.81,A -85,B 0,C 180,E1 1036.874,E2 1036.874} C_VEL
LIN {X 0,Y 751.606,Z 780.81,A -85,B 0,C 180,E1 1041.456,E2 1041.456} C_VEL
LIN {X 0,Y 751.579,Z 780.81,A -85,B 0,C 180,E1 1045.748,E2 1045.748} C_VEL
LIN {X 0,Y 751.709,Z 780.81,A -85,B 0,C 180,E1 1049.838,E2 1049.838} C_VEL
LIN {X 0,Y 751.661,Z 780.81,A -85,B 0,C 180,E1 1054.776,E2 1054.776} C_VEL
LIN {X 0,Y 751.675,Z 780.81,A -85,B 0,C 180,E1 1058.791,E2 1058.791} C_VEL
LIN {X 0,Y 751.704,Z 780.81,A -85,B 0,C 180,E1 1063.659,E2 1063.659} C_VEL
LIN {X 0,Y 751.598,Z 780.81,A -85,B 0,C 180,E1 1068.405,E2 1068.405} C_VEL
LIN {X 0,Y 751.641,Z 780.81,A -85,B 0,C 180,E1 1071.913,E2 1071.913} C_VEL
LIN {X 0,Y 751.84,Z 780.81,A -85,B 0,C 180,E1 1076.546,E2 1076.546} C_VEL
LIN {X 0,Y 751.956,Z 780.81,A -85,B 0,C 180,E1 1081.153,E2 1081.153} C_VEL
LIN {X 0,Y 751.739,Z 780.81,A -85,B 0,C 180,E1 1085.769,E2 1085.769} C_VEL
LIN {X 0,Y 751.651,Z 780.81,A -85,B 0,C 180,E1 1090.424,E2 1090.424} C_VEL
LIN {X 0,Y 751.601,Z 780.81,A -85,B 0,C 180,E1 1093.96,E2 1093.96} C_VEL
LIN {X 0,Y 751.644,Z 780.81,A -85,B 0,C 180,E1 1097.55,E2 1097.55} C_VEL
LIN {X 0,Y 751.583,Z 780.81,A -85,B 0,C 180,E1 1101.215,E2 1101.215} C_VEL
LIN {X 0,Y 751.549,Z 780.81,A -85,B 0,C 180,E1 1105.206,E2 1105.206} C_VEL
LIN {X 0,Y 751.713,Z 780.81,A -85,B 0,C 180,E1 1108.842,E2 1108.842} C_VEL
LIN {X 0,Y 751.837,Z 780.81,A -85,B 0,C 180,E1 1112.861,E2 1112.861} C_VEL
LIN {X 0,Y 751.774,Z 780.81,A -85,B 0,C 180,E1 1117.081,E2 1117.081} C_VEL
LIN {X 0,Y 751.756,Z 780.81,A -85,B 0,C 180,E1 1123.106,E2 1123.106} C_VEL
LIN {X 0,Y 751.353,Z 780.81,A -85,B 0,C 180,E1 1126.86,E2 1126.86} C_VEL
LIN {X 0,Y 751.742,Z 780.81,A -85,B 0,C 180,E1 1131.614,E2 1131.614} C_VEL
LIN {X 0,Y 751.834,Z 780.81,A -85,B 0,C 180,E1 1137.323,E2 1137.323} C_VEL
LIN {X 0,Y 753.504,Z 790.967,A -85,B 0,C 180,E1 1137.516,E2 1137.516} C_VEL
LIN {X 0,Y 753.516,Z 839.921,A -85,B 0,C 180,E1 1138.323,E2 1138.323} C_VEL
LIN {X 0,Y 753.31,Z 884.028,A -85,B 0,C 180,E1 1139.559,E2 1139.559} C_VEL
LIN {X 0,Y 753.071,Z 925.661,A -85,B 0,C 180,E1 1141.212,E2 1141.212} C_VEL
LIN {X 0,Y 752.782,Z 965.932,A -85,B 0,C 180,E1 1143.337,E2 1143.337} C_VEL
LIN {X 0,Y 752.482,Z 1003.026,A -85,B 0,C 180,E1 1145.864,E2 1145.864} C_VEL
LIN {X 0,Y 752.227,Z 1036.665,A -85,B 0,C 180,E1 1148.803,E2 1148.803} C_VEL
LIN {X 0,Y 751.989,Z 1065.076,A -85,B 0,C 180,E1 1152.004,E2 1152.004} C_VEL
LIN {X 0,Y 751.872,Z 1086.241,A -85,B 0,C 180,E1 1155.153,E2 1155.153} C_VEL
LIN {X 0,Y 751.853,Z 1101.124,A -85,B 0,C 180,E1 1158.112,E2 1158.112} C_VEL
LIN {X 0,Y 751.808,Z 1112.061,A -85,B 0,C 180,E1 1161.33,E2 1161.33} C_VEL
LIN {X 0,Y 751.849,Z 1117.747,A -85,B 0,C 180,E1 1164.233,E2 1164.233} C_VEL
LIN {X 0,Y 751.843,Z 1119.291,A -85,B 0,C 180,E1 1167.697,E2 1167.697} C_VEL
LIN {X 0,Y 751.886,Z 1115.344,A -85,B 0,C 180,E1 1171.152,E2 1171.152} C_VEL
LIN {X 0,Y 751.866,Z 1105.795,A -85,B 0,C 180,E1 1174.612,E2 1174.612} C_VEL
LIN {X 0,Y 751.87,Z 1090.021,A -85,B 0,C 180,E1 1178.088,E2 1178.088} C_VEL
LIN {X 0,Y 752.004,Z 1070.621,A -85,B 0,C 180,E1 1181.152,E2 1181.152} C_VEL
LIN {X 0,Y 752.118,Z 1045.031,A -85,B 0,C 180,E1 1184.249,E2 1184.249} C_VEL
LIN {X 0,Y 752.382,Z 1014.006,A -85,B 0,C 180,E1 1187.167,E2 1187.167} C_VEL
LIN {X 0,Y 752.697,Z 977.364,A -85,B 0,C 180,E1 1189.861,E2 1189.861} C_VEL
LIN {X 0,Y 753.036,Z 936.587,A -85,B 0,C 180,E1 1192.18,E2 1192.18} C_VEL
LIN {X 0,Y 753.312,Z 894.6,A -85,B 0,C 180,E1 1193.979,E2 1193.979} C_VEL
LIN {X 0,Y 753.535,Z 854.345,A -85,B 0,C 180,E1 1195.234,E2 1195.234} C_VEL
LIN {X 0,Y 753.751,Z 809.646,A -85,B 0,C 180,E1 1196.144,E2 1196.144} C_VEL
LIN {X 0,Y 752.065,Z 780.81,A -85,B 0,C 180,E1 1196.586,E2 1196.586} C_VEL
LIN {X 0,Y 751.845,Z 780.81,A -85,B 0,C 180,E1 1202.866,E2 1202.866} C_VEL
LIN {X 0,Y 751.757,Z 780.81,A -85,B 0,C 180,E1 1207.088,E2 1207.088} C_VEL
LIN {X 0,Y 751.775,Z 780.81,A -85,B 0,C 180,E1 1213.112,E2 1213.112} C_VEL
LIN {X 0,Y 751.364,Z 780.81,A -85,B 0,C 180,E1 1216.866,E2 1216.866} C_VEL
LIN {X 0,Y 751.557,Z 780.81,A -85,B 0,C 180,E1 1221.448,E2 1221.448} C_VEL
LIN {X 0,Y 751.571,Z 780.81,A -85,B 0,C 180,E1 1225.743,E2 1225.743} C_VEL
LIN {X 0,Y 751.701,Z 780.81,A -85,B 0,C 180,E1 1229.834,E2 1229.834} C_VEL
LIN {X 0,Y 751.67,Z 780.81,A -85,B 0,C 180,E1 1234.777,E2 1234.777} C_VEL
LIN {X 0,Y 751.668,Z 780.81,A -85,B 0,C 180,E1 1238.787,E2 1238.787} C_VEL
LIN {X 0,Y 751.728,Z 780.81,A -85,B 0,C 180,E1 1243.656,E2 1243.656} C_VEL
LIN {X 0,Y 751.629,Z 780.81,A -85,B 0,C 180,E1 1248.402,E2 1248.402} C_VEL
LIN {X 0,Y 751.939,Z 780.81,A -85,B 0,C 180,E1 1253.074,E2 1253.074} C_VEL
LIN {X 0,Y 751.74,Z 780.81,A -85,B 0,C 180,E1 1258.308,E2 1258.308} C_VEL
LIN {X 0,Y 747.747,Z 780.81,A -85,B 0,C 180,E1 1259.614,E2 1259.614} C_VEL
LIN {X 0,Y 744.021,Z 780.81,A -85,B 0,C 180,E1 1260.934,E2 1260.934} C_VEL
LIN {X 0,Y 743.834,Z 780.81,A -85,B 0,C 180,E1 1265.827,E2 1265.827} C_VEL
LIN {X 0,Y 743.736,Z 780.81,A -85,B 0,C 180,E1 1270.533,E2 1270.533} C_VEL
LIN {X 0,Y 743.854,Z 780.81,A -85,B 0,C 180,E1 1275.308,E2 1275.308} C_VEL
LIN {X 0,Y 743.902,Z 780.81,A -85,B 0,C 180,E1 1280.196,E2 1280.196} C_VEL
LIN {X 0,Y 743.723,Z 780.81,A -85,B 0,C 180,E1 1285.25,E2 1285.25} C_VEL
LIN {X 0,Y 743.749,Z 780.81,A -85,B 0,C 180,E1 1289.177,E2 1289.177} C_VEL
LIN {X 0,Y 743.772,Z 780.81,A -85,B 0,C 180,E1 1293.592,E2 1293.592} C_VEL
LIN {X 0,Y 743.723,Z 780.81,A -85,B 0,C 180,E1 1297.588,E2 1297.588} C_VEL
LIN {X 0,Y 743.702,Z 780.81,A -85,B 0,C 180,E1 1302.989,E2 1302.989} C_VEL
LIN {X 0,Y 743.738,Z 780.81,A -85,B 0,C 180,E1 1307.895,E2 1307.895} C_VEL
LIN {X 0,Y 743.723,Z 780.81,A -85,B 0,C 180,E1 1313.897,E2 1313.897} C_VEL
LIN {X 0,Y 743.813,Z 780.81,A -85,B 0,C 180,E1 1318.548,E2 1318.548} C_VEL
LIN {X 0,Y 743.959,Z 781.193,A -85,B 0,C 180,E1 1319.601,E2 1319.601} C_VEL
LIN {X 0,Y 746.347,Z 790.134,A -85,B 0,C 180,E1 1319.806,E2 1319.806} C_VEL
LIN {X 0,Y 746.665,Z 862.966,A -85,B 0,C 180,E1 1320.732,E2 1320.732} C_VEL
LIN {X 0,Y 746.435,Z 904.489,A -85,B 0,C 180,E1 1321.71,E2 1321.71} C_VEL
LIN {X 0,Y 746.041,Z 946.036,A -85,B 0,C 180,E1 1323.132,E2 1323.132} C_VEL
LIN {X 0,Y 745.554,Z 989.116,A -85,B 0,C 180,E1 1325.165,E2 1325.165} C_VEL
LIN {X 0,Y 745.05,Z 1027.896,A -85,B 0,C 180,E1 1327.569,E2 1327.569} C_VEL
LIN {X 0,Y 744.59,Z 1060.827,A -85,B 0,C 180,E1 1330.167,E2 1330.167} C_VEL
LIN {X 0,Y 744.325,Z 1089.384,A -85,B 0,C 180,E1 1333.004,E2 1333.004} C_VEL
LIN {X 0,Y 744.148,Z 1113.496,A -85,B 0,C 180,E1 1336.046,E2 1336.046} C_VEL
LIN {X 0,Y 743.949,Z 1132.222,A -85,B 0,C 180,E1 1339.17,E2 1339.17} C_VEL
LIN {X 0,Y 743.961,Z 1146.298,A -85,B 0,C 180,E1 1342.413,E2 1342.413} C_VEL
LIN {X 0,Y 743.984,Z 1154.484,A -85,B 0,C 180,E1 1345.339,E2 1345.339} C_VEL
LIN {X 0,Y 743.911,Z 1159.171,A -85,B 0,C 180,E1 1348.835,E2 1348.835} C_VEL
LIN {X 0,Y 743.912,Z 1158.226,A -85,B 0,C 180,E1 1352.328,E2 1352.328} C_VEL
LIN {X 0,Y 743.97,Z 1151.678,A -85,B 0,C 180,E1 1355.828,E2 1355.828} C_VEL
LIN {X 0,Y 743.987,Z 1140.637,A -85,B 0,C 180,E1 1359.056,E2 1359.056} C_VEL
LIN {X 0,Y 744.076,Z 1123.985,A -85,B 0,C 180,E1 1362.312,E2 1362.312} C_VEL
LIN {X 0,Y 744.272,Z 1103.54,A -85,B 0,C 180,E1 1365.303,E2 1365.303} C_VEL
LIN {X 0,Y 744.529,Z 1075.244,A -85,B 0,C 180,E1 1368.489,E2 1368.489} C_VEL
LIN {X 0,Y 744.918,Z 1041.717,A -85,B 0,C 180,E1 1371.415,E2 1371.415} C_VEL
LIN {X 0,Y 745.404,Z 1003.942,A -85,B 0,C 180,E1 1373.989,E2 1373.989} C_VEL
LIN {X 0,Y 745.827,Z 963.881,A -85,B 0,C 180,E1 1376.097,E2 1376.097} C_VEL
LIN {X 0,Y 746.3,Z 921.701,A -85,B 0,C 180,E1 1377.755,E2 1377.755} C_VEL
LIN {X 0,Y 746.693,Z 880.659,A -85,B 0,C 180,E1 1378.903,E2 1378.903} C_VEL
LIN {X 0,Y 746.836,Z 838.038,A -85,B 0,C 180,E1 1379.639,E2 1379.639} C_VEL
LIN {X 0,Y 745.622,Z 785.586,A -85,B 0,C 180,E1 1380.276,E2 1380.276} C_VEL
LIN {X 0,Y 744.003,Z 780.81,A -85,B 0,C 180,E1 1380.431,E2 1380.431} C_VEL
LIN {X 0,Y 743.603,Z 780.81,A -85,B 0,C 180,E1 1385.641,E2 1385.641} C_VEL
LIN {X 0,Y 743.487,Z 780.81,A -85,B 0,C 180,E1 1390.57,E2 1390.57} C_VEL
LIN {X 0,Y 743.901,Z 780.81,A -85,B 0,C 180,E1 1394.699,E2 1394.699} C_VEL
LIN {X 0,Y 743.694,Z 780.81,A -85,B 0,C 180,E1 1400.969,E2 1400.969} C_VEL
LIN {X 0,Y 743.696,Z 780.81,A -85,B 0,C 180,E1 1405.333,E2 1405.333} C_VEL
LIN {X 0,Y 743.751,Z 780.81,A -85,B 0,C 180,E1 1409.482,E2 1409.482} C_VEL
LIN {X 0,Y 743.794,Z 780.81,A -85,B 0,C 180,E1 1414.752,E2 1414.752} C_VEL
LIN {X 0,Y 743.722,Z 780.81,A -85,B 0,C 180,E1 1419.167,E2 1419.167} C_VEL
LIN {X 0,Y 743.798,Z 780.81,A -85,B 0,C 180,E1 1423.48,E2 1423.48} C_VEL
LIN {X 0,Y 743.678,Z 780.81,A -85,B 0,C 180,E1 1428.28,E2 1428.28} C_VEL
LIN {X 0,Y 743.998,Z 780.81,A -85,B 0,C 180,E1 1433.003,E2 1433.003} C_VEL
LIN {X 0,Y 743.953,Z 780.81,A -85,B 0,C 180,E1 1437.674,E2 1437.674} C_VEL
LIN {X 0,Y 743.801,Z 780.81,A -85,B 0,C 180,E1 1442.33,E2 1442.33} C_VEL
LIN {X 0,Y 743.84,Z 780.81,A -85,B 0,C 180,E1 1445.831,E2 1445.831} C_VEL
LIN {X 0,Y 743.749,Z 780.81,A -85,B 0,C 180,E1 1450.536,E2 1450.536} C_VEL
LIN {X 0,Y 743.866,Z 780.81,A -85,B 0,C 180,E1 1455.312,E2 1455.312} C_VEL
LIN {X 0,Y 743.726,Z 780.81,A -85,B 0,C 180,E1 1460.834,E2 1460.834} C_VEL
LIN {X 0,Y 743.671,Z 780.81,A -85,B 0,C 180,E1 1465.256,E2 1465.256} C_VEL
LIN {X 0,Y 743.749,Z 780.81,A -85,B 0,C 180,E1 1469.181,E2 1469.181} C_VEL
LIN {X 0,Y 743.746,Z 780.81,A -85,B 0,C 180,E1 1473.591,E2 1473.591} C_VEL
LIN {X 0,Y 743.699,Z 780.81,A -85,B 0,C 180,E1 1477.588,E2 1477.588} C_VEL
LIN {X 0,Y 743.856,Z 780.81,A -85,B 0,C 180,E1 1483.678,E2 1483.678} C_VEL
LIN {X 0,Y 743.462,Z 780.81,A -85,B 0,C 180,E1 1488.758,E2 1488.758} C_VEL
LIN {X 0,Y 743.84,Z 780.81,A -85,B 0,C 180,E1 1492.451,E2 1492.451} C_VEL
LIN {X 0,Y 743.859,Z 781.457,A -85,B 0,C 180,E1 1496.992,E2 1496.992} C_VEL
LIN {X 0,Y 746.626,Z 791.016,A -85,B 0,C 180,E1 1497.218,E2 1497.218} C_VEL
LIN {X 0,Y 746.519,Z 839.816,A -85,B 0,C 180,E1 1498.027,E2 1498.027} C_VEL
LIN {X 0,Y 746.173,Z 883.92,A -85,B 0,C 180,E1 1499.27,E2 1499.27} C_VEL
LIN {X 0,Y 745.768,Z 924.877,A -85,B 0,C 180,E1 1500.903,E2 1500.903} C_VEL
LIN {X 0,Y 745.359,Z 965.433,A -85,B 0,C 180,E1 1503.056,E2 1503.056} C_VEL
LIN {X 0,Y 744.888,Z 1003.196,A -85,B 0,C 180,E1 1505.653,E2 1505.653} C_VEL
LIN {X 0,Y 744.501,Z 1036.324,A -85,B 0,C 180,E1 1508.572,E2 1508.572} C_VEL
LIN {X 0,Y 744.202,Z 1064.809,A -85,B 0,C 180,E1 1511.809,E2 1511.809} C_VEL
LIN {X 0,Y 744.013,Z 1086.043,A -85,B 0,C 180,E1 1514.993,E2 1514.993} C_VEL
LIN {X 0,Y 743.977,Z 1100.994,A -85,B 0,C 180,E1 1517.984,E2 1517.984} C_VEL
LIN {X 0,Y 743.923,Z 1111.974,A -85,B 0,C 180,E1 1521.238,E2 1521.238} C_VEL
LIN {X 0,Y 743.922,Z 1117.991,A -85,B 0,C 180,E1 1524.373,E2 1524.373} C_VEL
LIN {X 0,Y 743.942,Z 1119.3,A -85,B 0,C 180,E1 1527.672,E2 1527.672} C_VEL
LIN {X 0,Y 743.984,Z 1115.411,A -85,B 0,C 180,E1 1531.164,E2 1531.164} C_VEL
LIN {X 0,Y 743.966,Z 1105.909,A -85,B 0,C 180,E1 1534.661,E2 1534.661} C_VEL
LIN {X 0,Y 744.051,Z 1091.721,A -85,B 0,C 180,E1 1537.88,E2 1537.88} C_VEL
LIN {X 0,Y 744.175,Z 1071.949,A -85,B 0,C 180,E1 1541.123,E2 1541.123} C_VEL
LIN {X 0,Y 744.358,Z 1046.745,A -85,B 0,C 180,E1 1544.25,E2 1544.25} C_VEL
LIN {X 0,Y 744.73,Z 1014.89,A -85,B 0,C 180,E1 1547.307,E2 1547.307} C_VEL
LIN {X 0,Y 745.19,Z 977.626,A -85,B 0,C 180,E1 1550.088,E2 1550.088} C_VEL
LIN {X 0,Y 745.704,Z 937.267,A -85,B 0,C 180,E1 1552.41,E2 1552.41} C_VEL
LIN {X 0,Y 746.159,Z 894.652,A -85,B 0,C 180,E1 1554.257,E2 1554.257} C_VEL
LIN {X 0,Y 746.538,Z 853.75,A -85,B 0,C 180,E1 1555.539,E2 1555.539} C_VEL
LIN {X 0,Y 746.849,Z 810.143,A -85,B 0,C 180,E1 1556.432,E2 1556.432} C_VEL
LIN {X 0,Y 745.24,Z 785.244,A -85,B 0,C 180,E1 1556.815,E2 1556.815} C_VEL
LIN {X 0,Y 744.073,Z 780.81,A -85,B 0,C 180,E1 1556.953,E2 1556.953} C_VEL
LIN {X 0,Y 743.806,Z 780.81,A -85,B 0,C 180,E1 1563.267,E2 1563.267} C_VEL
LIN {X 0,Y 743.683,Z 780.81,A -85,B 0,C 180,E1 1567.595,E2 1567.595} C_VEL
LIN {X 0,Y 743.866,Z 780.81,A -85,B 0,C 180,E1 1573.685,E2 1573.685} C_VEL
LIN {X 0,Y 743.462,Z 780.81,A -85,B 0,C 180,E1 1578.768,E2 1578.768} C_VEL
LIN {X 0,Y 743.492,Z 780.81,A -85,B 0,C 180,E1 1582.435,E2 1582.435} C_VEL
LIN {X 0,Y 743.53,Z 780.81,A -85,B 0,C 180,E1 1586.724,E2 1586.724} C_VEL
LIN {X 0,Y 743.671,Z 780.81,A -85,B 0,C 180,E1 1590.897,E2 1590.897} C_VEL
LIN {X 0,Y 743.804,Z 780.81,A -85,B 0,C 180,E1 1594.749,E2 1594.749} C_VEL
LIN {X 0,Y 743.704,Z 780.81,A -85,B 0,C 180,E1 1599.175,E2 1599.175} C_VEL
LIN {X 0,Y 743.817,Z 780.81,A -85,B 0,C 180,E1 1603.477,E2 1603.477} C_VEL
LIN {X 0,Y 743.707,Z 780.81,A -85,B 0,C 180,E1 1608.277,E2 1608.277} C_VEL
LIN {X 0,Y 744.01,Z 780.81,A -85,B 0,C 180,E1 1613.139,E2 1613.139} C_VEL
LIN {X 0,Y 743.838,Z 780.81,A -85,B 0,C 180,E1 1618.301,E2 1618.301} C_VEL
LIN {X 0,Y 744.021,Z 780.81,A -85,B 0,C 180,E1 1620.934,E2 1620.934} C_VEL
LIN {X 0,Y 741.536,Z 780.81,A -85,B 0,C 180,E1 1621.925,E2 1621.925} C_VEL
LIN {X 0,Y 736.025,Z 780.81,A -85,B 0,C 180,E1 1623.403,E2 1623.403} C_VEL
LIN {X 0,Y 735.937,Z 780.81,A -85,B 0,C 180,E1 1623.574,E2 1623.574} C_VEL
LIN {X 0,Y 736.039,Z 780.81,A -85,B 0,C 180,E1 1628.259,E2 1628.259} C_VEL
LIN {X 0,Y 735.964,Z 780.81,A -85,B 0,C 180,E1 1633.049,E2 1633.049} C_VEL
LIN {X 0,Y 735.826,Z 780.81,A -85,B 0,C 180,E1 1637.936,E2 1637.936} C_VEL
LIN {X 0,Y 735.799,Z 780.81,A -85,B 0,C 180,E1 1642.456,E2 1642.456} C_VEL
LIN {X 0,Y 735.759,Z 780.81,A -85,B 0,C 180,E1 1646.855,E2 1646.855} C_VEL
LIN {X 0,Y 735.914,Z 780.81,A -85,B 0,C 180,E1 1652.259,E2 1652.259} C_VEL
LIN {X 0,Y 735.779,Z 780.81,A -85,B 0,C 180,E1 1656.777,E2 1656.777} C_VEL
LIN {X 0,Y 735.792,Z 780.81,A -85,B 0,C 180,E1 1662.655,E2 1662.655} C_VEL
LIN {X 0,Y 735.824,Z 780.81,A -85,B 0,C 180,E1 1667.659,E2 1667.659} C_VEL
LIN {X 0,Y 735.765,Z 780.81,A -85,B 0,C 180,E1 1673.444,E2 1673.444} C_VEL
LIN {X 0,Y 735.878,Z 780.81,A -85,B 0,C 180,E1 1677.73,E2 1677.73} C_VEL
LIN {X 0,Y 735.982,Z 780.81,A -85,B 0,C 180,E1 1679.22,E2 1679.22} C_VEL
LIN {X 0,Y 739.546,Z 791.207,A -85,B 0,C 180,E1 1679.511,E2 1679.511} C_VEL
LIN {X 0,Y 739.775,Z 862.967,A -85,B 0,C 180,E1 1680.433,E2 1680.433} C_VEL
LIN {X 0,Y 739.408,Z 904.45,A -85,B 0,C 180,E1 1681.415,E2 1681.415} C_VEL
LIN {X 0,Y 738.827,Z 947.442,A -85,B 0,C 180,E1 1682.909,E2 1682.909} C_VEL
LIN {X 0,Y 738.186,Z 989.952,A -85,B 0,C 180,E1 1684.945,E2 1684.945} C_VEL
LIN {X 0,Y 737.514,Z 1030.08,A -85,B 0,C 180,E1 1687.48,E2 1687.48} C_VEL
LIN {X 0,Y 736.86,Z 1066.102,A -85,B 0,C 180,E1 1690.427,E2 1690.427} C_VEL
LIN {X 0,Y 736.482,Z 1096.258,A -85,B 0,C 180,E1 1693.612,E2 1693.612} C_VEL
LIN {X 0,Y 736.284,Z 1120.375,A -85,B 0,C 180,E1 1696.952,E2 1696.952} C_VEL
LIN {X 0,Y 736.104,Z 1137.365,A -85,B 0,C 180,E1 1700.118,E2 1700.118} C_VEL
LIN {X 0,Y 736.043,Z 1150.117,A -85,B 0,C 180,E1 1703.516,E2 1703.516} C_VEL
LIN {X 0,Y 735.991,Z 1156.665,A -85,B 0,C 180,E1 1706.468,E2 1706.468} C_VEL
LIN {X 0,Y 736.024,Z 1159.171,A -85,B 0,C 180,E1 1708.823,E2 1708.823} C_VEL
LIN {X 0,Y 736.012,Z 1158.227,A -85,B 0,C 180,E1 1712.353,E2 1712.353} C_VEL
LIN {X 0,Y 736.221,Z 1153.596,A -85,B 0,C 180,E1 1715.147,E2 1715.147} C_VEL
LIN {X 0,Y 736.18,Z 1142.959,A -85,B 0,C 180,E1 1718.558,E2 1718.558} C_VEL
LIN {X 0,Y 736.286,Z 1127.481,A -85,B 0,C 180,E1 1721.842,E2 1721.842} C_VEL
LIN {X 0,Y 736.485,Z 1105.022,A -85,B 0,C 180,E1 1725.28,E2 1725.28} C_VEL
LIN {X 0,Y 736.806,Z 1076.777,A -85,B 0,C 180,E1 1728.534,E2 1728.534} C_VEL
LIN {X 0,Y 737.34,Z 1042.816,A -85,B 0,C 180,E1 1731.562,E2 1731.562} C_VEL
LIN {X 0,Y 737.989,Z 1003.944,A -85,B 0,C 180,E1 1734.246,E2 1734.246} C_VEL
LIN {X 0,Y 738.648,Z 963.319,A -85,B 0,C 180,E1 1736.397,E2 1736.397} C_VEL
LIN {X 0,Y 739.248,Z 921.706,A -85,B 0,C 180,E1 1738.043,E2 1738.043} C_VEL
LIN {X 0,Y 739.74,Z 881.937,A -85,B 0,C 180,E1 1739.173,E2 1739.173} C_VEL
LIN {X 0,Y 739.983,Z 837.702,A -85,B 0,C 180,E1 1739.946,E2 1739.946} C_VEL
LIN {X 0,Y 738.951,Z 788.765,A -85,B 0,C 180,E1 1740.543,E2 1740.543} C_VEL
LIN {X 0,Y 736.041,Z 780.81,A -85,B 0,C 180,E1 1740.822,E2 1740.822} C_VEL
LIN {X 0,Y 735.662,Z 780.81,A -85,B 0,C 180,E1 1745.109,E2 1745.109} C_VEL
LIN {X 0,Y 735.515,Z 780.81,A -85,B 0,C 180,E1 1749.559,E2 1749.559} C_VEL
LIN {X 0,Y 736.011,Z 780.81,A -85,B 0,C 180,E1 1754.27,E2 1754.27} C_VEL
LIN {X 0,Y 735.842,Z 780.81,A -85,B 0,C 180,E1 1760.471,E2 1760.471} C_VEL
LIN {X 0,Y 735.814,Z 780.81,A -85,B 0,C 180,E1 1765.23,E2 1765.23} C_VEL
LIN {X 0,Y 735.748,Z 780.81,A -85,B 0,C 180,E1 1770.475,E2 1770.475} C_VEL
LIN {X 0,Y 735.903,Z 780.81,A -85,B 0,C 180,E1 1774.62,E2 1774.62} C_VEL
LIN {X 0,Y 735.787,Z 780.81,A -85,B 0,C 180,E1 1779.571,E2 1779.571} C_VEL
LIN {X 0,Y 735.899,Z 780.81,A -85,B 0,C 180,E1 1784.522,E2 1784.522} C_VEL
LIN {X 0,Y 735.983,Z 780.81,A -85,B 0,C 180,E1 1790.236,E2 1790.236} C_VEL
LIN {X 0,Y 736.002,Z 780.81,A -85,B 0,C 180,E1 1794.111,E2 1794.111} C_VEL
LIN {X 0,Y 735.88,Z 780.81,A -85,B 0,C 180,E1 1798.825,E2 1798.825} C_VEL
LIN {X 0,Y 735.918,Z 780.81,A -85,B 0,C 180,E1 1802.355,E2 1802.355} C_VEL
LIN {X 0,Y 735.93,Z 780.81,A -85,B 0,C 180,E1 1805.894,E2 1805.894} C_VEL
LIN {X 0,Y 735.854,Z 780.81,A -85,B 0,C 180,E1 1810.651,E2 1810.651} C_VEL
LIN {X 0,Y 735.971,Z 780.81,A -85,B 0,C 180,E1 1815.48,E2 1815.48} C_VEL
LIN {X 0,Y 735.908,Z 780.81,A -85,B 0,C 180,E1 1820.429,E2 1820.429} C_VEL
LIN {X 0,Y 735.743,Z 780.81,A -85,B 0,C 180,E1 1825.548,E2 1825.548} C_VEL
LIN {X 0,Y 735.727,Z 780.81,A -85,B 0,C 180,E1 1830.388,E2 1830.388} C_VEL
LIN {X 0,Y 735.689,Z 780.81,A -85,B 0,C 180,E1 1835.103,E2 1835.103} C_VEL
LIN {X 0,Y 735.459,Z 780.81,A -85,B 0,C 180,E1 1839.558,E2 1839.558} C_VEL
LIN {X 0,Y 735.948,Z 780.81,A -85,B 0,C 180,E1 1844.269,E2 1844.269} C_VEL
LIN {X 0,Y 735.871,Z 780.81,A -85,B 0,C 180,E1 1850.463,E2 1850.463} C_VEL
LIN {X 0,Y 735.702,Z 780.81,A -85,B 0,C 180,E1 1855.233,E2 1855.233} C_VEL
LIN {X 0,Y 735.826,Z 780.81,A -85,B 0,C 180,E1 1856.624,E2 1856.624} C_VEL
LIN {X 0,Y 739.775,Z 791.85,A -85,B 0,C 180,E1 1856.924,E2 1856.924} C_VEL
LIN {X 0,Y 739.564,Z 841.107,A -85,B 0,C 180,E1 1857.756,E2 1857.756} C_VEL
LIN {X 0,Y 739.073,Z 886.802,A -85,B 0,C 180,E1 1859.08,E2 1859.08} C_VEL
LIN {X 0,Y 738.487,Z 928.806,A -85,B 0,C 180,E1 1860.817,E2 1860.817} C_VEL
LIN {X 0,Y 737.867,Z 967.89,A -85,B 0,C 180,E1 1862.954,E2 1862.954} C_VEL
LIN {X 0,Y 737.281,Z 1004.378,A -85,B 0,C 180,E1 1865.519,E2 1865.519} C_VEL
LIN {X 0,Y 736.759,Z 1037.257,A -85,B 0,C 180,E1 1868.47,E2 1868.47} C_VEL
LIN {X 0,Y 736.403,Z 1064.53,A -85,B 0,C 180,E1 1871.61,E2 1871.61} C_VEL
LIN {X 0,Y 736.223,Z 1085.074,A -85,B 0,C 180,E1 1874.697,E2 1874.697} C_VEL
LIN {X 0,Y 736.118,Z 1100.926,A -85,B 0,C 180,E1 1877.87,E2 1877.87} C_VEL
LIN {X 0,Y 736.053,Z 1111.887,A -85,B 0,C 180,E1 1881.143,E2 1881.143} C_VEL
LIN {X 0,Y 736.066,Z 1117.653,A -85,B 0,C 180,E1 1884.109,E2 1884.109} C_VEL
LIN {X 0,Y 736.047,Z 1119.31,A -85,B 0,C 180,E1 1887.647,E2 1887.647} C_VEL
LIN {X 0,Y 736.092,Z 1115.478,A -85,B 0,C 180,E1 1891.177,E2 1891.177} C_VEL
LIN {X 0,Y 736.096,Z 1106.016,A -85,B 0,C 180,E1 1894.711,E2 1894.711} C_VEL
LIN {X 0,Y 736.165,Z 1091.894,A -85,B 0,C 180,E1 1897.965,E2 1897.965} C_VEL
LIN {X 0,Y 736.326,Z 1072.194,A -85,B 0,C 180,E1 1901.243,E2 1901.243} C_VEL
LIN {X 0,Y 736.596,Z 1047.065,A -85,B 0,C 180,E1 1904.402,E2 1904.402} C_VEL
LIN {X 0,Y 737.096,Z 1015.484,A -85,B 0,C 180,E1 1907.474,E2 1907.474} C_VEL
LIN {X 0,Y 737.682,Z 978.812,A -85,B 0,C 180,E1 1910.256,E2 1910.256} C_VEL
LIN {X 0,Y 738.375,Z 938.386,A -85,B 0,C 180,E1 1912.621,E2 1912.621} C_VEL
LIN {X 0,Y 739,Z 897.271,A -85,B 0,C 180,E1 1914.442,E2 1914.442} C_VEL
LIN {X 0,Y 739.53,Z 855.862,A -85,B 0,C 180,E1 1915.781,E2 1915.781} C_VEL
LIN {X 0,Y 739.933,Z 812.281,A -85,B 0,C 180,E1 1916.699,E2 1916.699} C_VEL
LIN {X 0,Y 738.515,Z 787.658,A -85,B 0,C 180,E1 1917.089,E2 1917.089} C_VEL
LIN {X 0,Y 736.162,Z 780.81,A -85,B 0,C 180,E1 1917.287,E2 1917.287} C_VEL
LIN {X 0,Y 735.868,Z 780.81,A -85,B 0,C 180,E1 1922.667,E2 1922.667} C_VEL
LIN {X 0,Y 735.661,Z 780.81,A -85,B 0,C 180,E1 1928.042,E2 1928.042} C_VEL
LIN {X 0,Y 735.895,Z 780.81,A -85,B 0,C 180,E1 1932.66,E2 1932.66} C_VEL
LIN {X 0,Y 735.524,Z 780.81,A -85,B 0,C 180,E1 1937.321,E2 1937.321} C_VEL
LIN {X 0,Y 735.586,Z 780.81,A -85,B 0,C 180,E1 1941.96,E2 1941.96} C_VEL
LIN {X 0,Y 735.682,Z 780.81,A -85,B 0,C 180,E1 1946.322,E2 1946.322} C_VEL
LIN {X 0,Y 735.757,Z 780.81,A -85,B 0,C 180,E1 1950.471,E2 1950.471} C_VEL
LIN {X 0,Y 735.9,Z 780.81,A -85,B 0,C 180,E1 1954.624,E2 1954.624} C_VEL
LIN {X 0,Y 735.776,Z 780.81,A -85,B 0,C 180,E1 1959.567,E2 1959.567} C_VEL
LIN {X 0,Y 735.926,Z 780.81,A -85,B 0,C 180,E1 1964.519,E2 1964.519} C_VEL
LIN {X 0,Y 736.038,Z 780.81,A -85,B 0,C 180,E1 1970.219,E2 1970.219} C_VEL
LIN {X 0,Y 736.042,Z 780.81,A -85,B 0,C 180,E1 1974.107,E2 1974.107} C_VEL
LIN {X 0,Y 735.917,Z 780.81,A -85,B 0,C 180,E1 1978.822,E2 1978.822} C_VEL
LIN {X 0,Y 735.912,Z 780.81,A -85,B 0,C 180,E1 1982.351,E2 1982.351} C_VEL
LIN {X 0,Y 735.937,Z 780.81,A -85,B 0,C 180,E1 1983.574,E2 1983.574} C_VEL
LIN {X 0,Y 734.715,Z 780.81,A -85,B 0,C 180,E1 1984.248,E2 1984.248} C_VEL
LIN {X 0,Y 728.101,Z 780.81,A -85,B 0,C 180,E1 1986.08,E2 1986.08} C_VEL
LIN {X 0,Y 727.993,Z 780.81,A -85,B 0,C 180,E1 1986.253,E2 1986.253} C_VEL
LIN {X 0,Y 727.944,Z 780.81,A -85,B 0,C 180,E1 1990.764,E2 1990.764} C_VEL
LIN {X 0,Y 728.054,Z 780.81,A -85,B 0,C 180,E1 1995.649,E2 1995.649} C_VEL
LIN {X 0,Y 727.952,Z 780.81,A -85,B 0,C 180,E1 2000.911,E2 2000.911} C_VEL
LIN {X 0,Y 727.839,Z 780.81,A -85,B 0,C 180,E1 2005.842,E2 2005.842} C_VEL
LIN {X 0,Y 727.858,Z 780.81,A -85,B 0,C 180,E1 2009.877,E2 2009.877} C_VEL
LIN {X 0,Y 727.885,Z 780.81,A -85,B 0,C 180,E1 2014.083,E2 2014.083} C_VEL
LIN {X 0,Y 727.688,Z 780.81,A -85,B 0,C 180,E1 2018.524,E2 2018.524} C_VEL
LIN {X 0,Y 727.744,Z 780.81,A -85,B 0,C 180,E1 2023.385,E2 2023.385} C_VEL
LIN {X 0,Y 727.785,Z 780.81,A -85,B 0,C 180,E1 2028.361,E2 2028.361} C_VEL
LIN {X 0,Y 727.838,Z 780.81,A -85,B 0,C 180,E1 2034.05,E2 2034.05} C_VEL
LIN {X 0,Y 728.063,Z 781.571,A -85,B 0,C 180,E1 2038.869,E2 2038.869} C_VEL
LIN {X 0,Y 732.731,Z 792.576,A -85,B 0,C 180,E1 2039.212,E2 2039.212} C_VEL
LIN {X 0,Y 732.884,Z 864.065,A -85,B 0,C 180,E1 2040.146,E2 2040.146} C_VEL
LIN {X 0,Y 732.369,Z 906.516,A -85,B 0,C 180,E1 2041.177,E2 2041.177} C_VEL
LIN {X 0,Y 731.647,Z 948.064,A -85,B 0,C 180,E1 2042.648,E2 2042.648} C_VEL
LIN {X 0,Y 730.877,Z 989.963,A -85,B 0,C 180,E1 2044.677,E2 2044.677} C_VEL
LIN {X 0,Y 730.007,Z 1029.668,A -85,B 0,C 180,E1 2047.206,E2 2047.206} C_VEL
LIN {X 0,Y 729.248,Z 1064.896,A -85,B 0,C 180,E1 2050.099,E2 2050.099} C_VEL
LIN {X 0,Y 728.717,Z 1094.959,A -85,B 0,C 180,E1 2053.278,E2 2053.278} C_VEL
LIN {X 0,Y 728.416,Z 1118.416,A -85,B 0,C 180,E1 2056.503,E2 2056.503} C_VEL
LIN {X 0,Y 728.185,Z 1135.647,A -85,B 0,C 180,E1 2059.623,E2 2059.623} C_VEL
LIN {X 0,Y 728.128,Z 1148.22,A -85,B 0,C 180,E1 2062.846,E2 2062.846} C_VEL
LIN {X 0,Y 728.167,Z 1155.684,A -85,B 0,C 180,E1 2065.834,E2 2065.834} C_VEL
LIN {X 0,Y 728.126,Z 1159.171,A -85,B 0,C 180,E1 2068.81,E2 2068.81} C_VEL
LIN {X 0,Y 728.107,Z 1158.227,A -85,B 0,C 180,E1 2072.378,E2 2072.378} C_VEL
LIN {X 0,Y 728.296,Z 1153.381,A -85,B 0,C 180,E1 2075.3,E2 2075.3} C_VEL
LIN {X 0,Y 728.254,Z 1141.811,A -85,B 0,C 180,E1 2078.952,E2 2078.952} C_VEL
LIN {X 0,Y 728.358,Z 1124.935,A -85,B 0,C 180,E1 2082.416,E2 2082.416} C_VEL
LIN {X 0,Y 728.634,Z 1103.537,A -85,B 0,C 180,E1 2085.64,E2 2085.64} C_VEL
LIN {X 0,Y 729.106,Z 1075.241,A -85,B 0,C 180,E1 2088.894,E2 2088.894} C_VEL
LIN {X 0,Y 729.756,Z 1041.719,A -85,B 0,C 180,E1 2091.883,E2 2091.883} C_VEL
LIN {X 0,Y 730.551,Z 1004.017,A -85,B 0,C 180,E1 2094.505,E2 2094.505} C_VEL
LIN {X 0,Y 731.43,Z 962.195,A -85,B 0,C 180,E1 2096.732,E2 2096.732} C_VEL
LIN {X 0,Y 732.199,Z 919.764,A -85,B 0,C 180,E1 2098.405,E2 2098.405} C_VEL
LIN {X 0,Y 732.807,Z 878.388,A -85,B 0,C 180,E1 2099.553,E2 2099.553} C_VEL
LIN {X 0,Y 733.145,Z 834.82,A -85,B 0,C 180,E1 2100.293,E2 2100.293} C_VEL
LIN {X 0,Y 731.895,Z 790.454,A -85,B 0,C 180,E1 2100.851,E2 2100.851} C_VEL
LIN {X 0,Y 728.097,Z 780.81,A -85,B 0,C 180,E1 2101.166,E2 2101.166} C_VEL
LIN {X 0,Y 727.768,Z 780.81,A -85,B 0,C 180,E1 2105.942,E2 2105.942} C_VEL
LIN {X 0,Y 727.865,Z 780.81,A -85,B 0,C 180,E1 2111.649,E2 2111.649} C_VEL
LIN {X 0,Y 727.963,Z 780.81,A -85,B 0,C 180,E1 2115.12,E2 2115.12} C_VEL
LIN {X 0,Y 727.914,Z 780.81,A -85,B 0,C 180,E1 2120.182,E2 2120.182} C_VEL
LIN {X 0,Y 727.799,Z 780.81,A -85,B 0,C 180,E1 2124.463,E2 2124.463} C_VEL
LIN {X 0,Y 727.889,Z 780.81,A -85,B 0,C 180,E1 2130.124,E2 2130.124} C_VEL
LIN {X 0,Y 727.987,Z 780.81,A -85,B 0,C 180,E1 2134.164,E2 2134.164} C_VEL
LIN {X 0,Y 727.879,Z 780.81,A -85,B 0,C 180,E1 2139.339,E2 2139.339} C_VEL
LIN {X 0,Y 727.982,Z 780.81,A -85,B 0,C 180,E1 2144.35,E2 2144.35} C_VEL
LIN {X 0,Y 728.157,Z 780.81,A -85,B 0,C 180,E1 2149.239,E2 2149.239} C_VEL
LIN {X 0,Y 728.1,Z 780.81,A -85,B 0,C 180,E1 2154.047,E2 2154.047} C_VEL
LIN {X 0,Y 727.981,Z 780.81,A -85,B 0,C 180,E1 2158.813,E2 2158.813} C_VEL
LIN {X 0,Y 728.016,Z 780.81,A -85,B 0,C 180,E1 2162.381,E2 2162.381} C_VEL
LIN {X 0,Y 728.037,Z 780.81,A -85,B 0,C 180,E1 2165.958,E2 2165.958} C_VEL
LIN {X 0,Y 727.951,Z 780.81,A -85,B 0,C 180,E1 2170.768,E2 2170.768} C_VEL
LIN {X 0,Y 728.062,Z 780.81,A -85,B 0,C 180,E1 2175.653,E2 2175.653} C_VEL
LIN {X 0,Y 727.914,Z 780.81,A -85,B 0,C 180,E1 2180.907,E2 2180.907} C_VEL
LIN {X 0,Y 727.804,Z 780.81,A -85,B 0,C 180,E1 2185.847,E2 2185.847} C_VEL
LIN {X 0,Y 727.86,Z 780.81,A -85,B 0,C 180,E1 2189.882,E2 2189.882} C_VEL
LIN {X 0,Y 727.865,Z 780.81,A -85,B 0,C 180,E1 2194.089,E2 2194.089} C_VEL
LIN {X 0,Y 727.644,Z 780.81,A -85,B 0,C 180,E1 2198.531,E2 2198.531} C_VEL
LIN {X 0,Y 727.964,Z 780.81,A -85,B 0,C 180,E1 2203.405,E2 2203.405} C_VEL
LIN {X 0,Y 727.619,Z 780.81,A -85,B 0,C 180,E1 2208.378,E2 2208.378} C_VEL
LIN {X 0,Y 727.944,Z 780.81,A -85,B 0,C 180,E1 2212.988,E2 2212.988} C_VEL
LIN {X 0,Y 727.907,Z 781.574,A -85,B 0,C 180,E1 2216.267,E2 2216.267} C_VEL
LIN {X 0,Y 732.946,Z 795.163,A -85,B 0,C 180,E1 2216.658,E2 2216.658} C_VEL
LIN {X 0,Y 732.636,Z 842.146,A -85,B 0,C 180,E1 2217.477,E2 2217.477} C_VEL
LIN {X 0,Y 731.981,Z 888.02,A -85,B 0,C 180,E1 2218.829,E2 2218.829} C_VEL
LIN {X 0,Y 731.208,Z 930.224,A -85,B 0,C 180,E1 2220.607,E2 2220.607} C_VEL
LIN {X 0,Y 730.466,Z 967.995,A -85,B 0,C 180,E1 2222.702,E2 2222.702} C_VEL
LIN {X 0,Y 729.762,Z 1003.443,A -85,B 0,C 180,E1 2225.21,E2 2225.21} C_VEL
LIN {X 0,Y 729.107,Z 1036.667,A -85,B 0,C 180,E1 2228.206,E2 2228.206} C_VEL
LIN {X 0,Y 728.645,Z 1064.252,A -85,B 0,C 180,E1 2231.407,E2 2231.407} C_VEL
LIN {X 0,Y 728.373,Z 1085.441,A -85,B 0,C 180,E1 2234.627,E2 2234.627} C_VEL
LIN {X 0,Y 728.288,Z 1100.124,A -85,B 0,C 180,E1 2237.586,E2 2237.586} C_VEL
LIN {X 0,Y 728.167,Z 1111.8,A -85,B 0,C 180,E1 2241.047,E2 2241.047} C_VEL
LIN {X 0,Y 728.188,Z 1117.606,A -85,B 0,C 180,E1 2244.045,E2 2244.045} C_VEL
LIN {X 0,Y 728.146,Z 1119.319,A -85,B 0,C 180,E1 2247.622,E2 2247.622} C_VEL
LIN {X 0,Y 728.191,Z 1115.545,A -85,B 0,C 180,E1 2251.19,E2 2251.19} C_VEL
LIN {X 0,Y 728.198,Z 1106.123,A -85,B 0,C 180,E1 2254.762,E2 2254.762} C_VEL
LIN {X 0,Y 728.299,Z 1092.067,A -85,B 0,C 180,E1 2258.052,E2 2258.052} C_VEL
LIN {X 0,Y 728.5,Z 1072.436,A -85,B 0,C 180,E1 2261.366,E2 2261.366} C_VEL
LIN {X 0,Y 728.89,Z 1046.335,A -85,B 0,C 180,E1 2264.677,E2 2264.677} C_VEL
LIN {X 0,Y 729.484,Z 1014.095,A -85,B 0,C 180,E1 2267.823,E2 2267.823} C_VEL
LIN {X 0,Y 730.253,Z 977.518,A -85,B 0,C 180,E1 2270.597,E2 2270.597} C_VEL
LIN {X 0,Y 731.116,Z 937.264,A -85,B 0,C 180,E1 2272.955,E2 2272.955} C_VEL
LIN {X 0,Y 731.892,Z 895.397,A -85,B 0,C 180,E1 2274.806,E2 2274.806} C_VEL
LIN {X 0,Y 732.559,Z 854.075,A -85,B 0,C 180,E1 2276.128,E2 2276.128} C_VEL
LIN {X 0,Y 733.075,Z 809.72,A -85,B 0,C 180,E1 2277.05,E2 2277.05} C_VEL
LIN {X 0,Y 731.639,Z 789.73,A -85,B 0,C 180,E1 2277.379,E2 2277.379} C_VEL
LIN {X 0,Y 728.21,Z 780.81,A -85,B 0,C 180,E1 2277.699,E2 2277.699} C_VEL
LIN {X 0,Y 727.969,Z 780.81,A -85,B 0,C 180,E1 2282.664,E2 2282.664} C_VEL
LIN {X 0,Y 727.754,Z 780.81,A -85,B 0,C 180,E1 2287.915,E2 2287.915} C_VEL
LIN {X 0,Y 727.973,Z 780.81,A -85,B 0,C 180,E1 2293.412,E2 2293.412} C_VEL
LIN {X 0,Y 727.635,Z 780.81,A -85,B 0,C 180,E1 2298.386,E2 2298.386} C_VEL
LIN {X 0,Y 727.681,Z 780.81,A -85,B 0,C 180,E1 2302.976,E2 2302.976} C_VEL
LIN {X 0,Y 727.716,Z 780.81,A -85,B 0,C 180,E1 2307.328,E2 2307.328} C_VEL
LIN {X 0,Y 727.818,Z 780.81,A -85,B 0,C 180,E1 2311.479,E2 2311.479} C_VEL
LIN {X 0,Y 727.847,Z 780.81,A -85,B 0,C 180,E1 2315.995,E2 2315.995} C_VEL
LIN {X 0,Y 727.925,Z 780.81,A -85,B 0,C 180,E1 2320.602,E2 2320.602} C_VEL
LIN {X 0,Y 728.003,Z 780.81,A -85,B 0,C 180,E1 2325.577,E2 2325.577} C_VEL
LIN {X 0,Y 728.102,Z 780.81,A -85,B 0,C 180,E1 2330.443,E2 2330.443} C_VEL
LIN {X 0,Y 728,Z 780.81,A -85,B 0,C 180,E1 2335.236,E2 2335.236} C_VEL
LIN {X 0,Y 728.1,Z 780.81,A -85,B 0,C 180,E1 2339.998,E2 2339.998} C_VEL
LIN {X 0,Y 728.155,Z 780.81,A -85,B 0,C 180,E1 2345.041,E2 2345.041} C_VEL
LIN {X 0,Y 727.993,Z 780.81,A -85,B 0,C 180,E1 2346.253,E2 2346.253} C_VEL
LIN {X 0,Y 724.061,Z 780.81,A -85,B 0,C 180,E1 2347.595,E2 2347.595} C_VEL
LIN {X 0,Y 720.148,Z 780.81,A -85,B 0,C 180,E1 2348.951,E2 2348.951} C_VEL
LIN {X 0,Y 720.109,Z 780.81,A -85,B 0,C 180,E1 2353.342,E2 2353.342} C_VEL
LIN {X 0,Y 720.04,Z 780.81,A -85,B 0,C 180,E1 2358.343,E2 2358.343} C_VEL
LIN {X 0,Y 720.046,Z 780.81,A -85,B 0,C 180,E1 2363.493,E2 2363.493} C_VEL
LIN {X 0,Y 719.986,Z 780.81,A -85,B 0,C 180,E1 2368.856,E2 2368.856} C_VEL
LIN {X 0,Y 720.052,Z 780.81,A -85,B 0,C 180,E1 2373.06,E2 2373.06} C_VEL
LIN {X 0,Y 719.904,Z 780.81,A -85,B 0,C 180,E1 2377.487,E2 2377.487} C_VEL
LIN {X 0,Y 719.818,Z 780.81,A -85,B 0,C 180,E1 2382.713,E2 2382.713} C_VEL
LIN {X 0,Y 719.849,Z 780.81,A -85,B 0,C 180,E1 2387.797,E2 2387.797} C_VEL
LIN {X 0,Y 719.933,Z 780.81,A -85,B 0,C 180,E1 2392.886,E2 2392.886} C_VEL
LIN {X 0,Y 720.093,Z 780.81,A -85,B 0,C 180,E1 2398.466,E2 2398.466} C_VEL
LIN {X 0,Y 726.046,Z 796.06,A -85,B 0,C 180,E1 2398.937,E2 2398.937} C_VEL
LIN {X 0,Y 726.008,Z 864.067,A -85,B 0,C 180,E1 2399.834,E2 2399.834} C_VEL
LIN {X 0,Y 725.389,Z 907.036,A -85,B 0,C 180,E1 2400.889,E2 2400.889} C_VEL
LIN {X 0,Y 724.47,Z 949.163,A -85,B 0,C 180,E1 2402.403,E2 2402.403} C_VEL
LIN {X 0,Y 723.533,Z 989.957,A -85,B 0,C 180,E1 2404.401,E2 2404.401} C_VEL
LIN {X 0,Y 722.478,Z 1029.465,A -85,B 0,C 180,E1 2406.94,E2 2406.94} C_VEL
LIN {X 0,Y 721.604,Z 1063.866,A -85,B 0,C 180,E1 2409.785,E2 2409.785} C_VEL
LIN {X 0,Y 720.968,Z 1093.634,A -85,B 0,C 180,E1 2412.936,E2 2412.936} C_VEL
LIN {X 0,Y 720.609,Z 1116.455,A -85,B 0,C 180,E1 2416.045,E2 2416.045} C_VEL
LIN {X 0,Y 720.317,Z 1135.271,A -85,B 0,C 180,E1 2419.422,E2 2419.422} C_VEL
LIN {X 0,Y 720.238,Z 1148.22,A -85,B 0,C 180,E1 2422.768,E2 2422.768} C_VEL
LIN {X 0,Y 720.284,Z 1155.684,A -85,B 0,C 180,E1 2425.788,E2 2425.788} C_VEL
LIN {X 0,Y 720.243,Z 1159.17,A -85,B 0,C 180,E1 2428.797,E2 2428.797} C_VEL
LIN {X 0,Y 720.203,Z 1158.226,A -85,B 0,C 180,E1 2432.404,E2 2432.404} C_VEL
LIN {X 0,Y 720.383,Z 1153.381,A -85,B 0,C 180,E1 2435.358,E2 2435.358} C_VEL
LIN {X 0,Y 720.364,Z 1141.811,A -85,B 0,C 180,E1 2439.051,E2 2439.051} C_VEL
LIN {X 0,Y 720.487,Z 1125.242,A -85,B 0,C 180,E1 2442.5,E2 2442.5} C_VEL
LIN {X 0,Y 720.838,Z 1105.493,A -85,B 0,C 180,E1 2445.555,E2 2445.555} C_VEL
LIN {X 0,Y 721.372,Z 1076.893,A -85,B 0,C 180,E1 2448.934,E2 2448.934} C_VEL
LIN {X 0,Y 722.168,Z 1043.635,A -85,B 0,C 180,E1 2451.97,E2 2451.97} C_VEL
LIN {X 0,Y 723.14,Z 1005.099,A -85,B 0,C 180,E1 2454.703,E2 2454.703} C_VEL
LIN {X 0,Y 724.182,Z 964.539,A -85,B 0,C 180,E1 2456.906,E2 2456.906} C_VEL
LIN {X 0,Y 725.069,Z 925.183,A -85,B 0,C 180,E1 2458.519,E2 2458.519} C_VEL
LIN {X 0,Y 725.874,Z 882.92,A -85,B 0,C 180,E1 2459.761,E2 2459.761} C_VEL
LIN {X 0,Y 726.276,Z 841.317,A -85,B 0,C 180,E1 2460.523,E2 2460.523} C_VEL
LIN {X 0,Y 725.338,Z 793.555,A -85,B 0,C 180,E1 2461.125,E2 2461.125} C_VEL
LIN {X 0,Y 720.175,Z 780.81,A -85,B 0,C 180,E1 2461.576,E2 2461.576} C_VEL
LIN {X 0,Y 719.877,Z 780.81,A -85,B 0,C 180,E1 2467.498,E2 2467.498} C_VEL
LIN {X 0,Y 720.059,Z 780.81,A -85,B 0,C 180,E1 2472.748,E2 2472.748} C_VEL
LIN {X 0,Y 719.724,Z 780.81,A -85,B 0,C 180,E1 2477.801,E2 2477.801} C_VEL
LIN {X 0,Y 719.855,Z 780.81,A -85,B 0,C 180,E1 2482.909,E2 2482.909} C_VEL
LIN {X 0,Y 719.803,Z 780.81,A -85,B 0,C 180,E1 2487.11,E2 2487.11} C_VEL
LIN {X 0,Y 719.926,Z 780.81,A -85,B 0,C 180,E1 2491.831,E2 2491.831} C_VEL
LIN {X 0,Y 719.983,Z 780.81,A -85,B 0,C 180,E1 2496.505,E2 2496.505} C_VEL
LIN {X 0,Y 720.076,Z 780.81,A -85,B 0,C 180,E1 2501.658,E2 2501.658} C_VEL
LIN {X 0,Y 719.979,Z 780.81,A -85,B 0,C 180,E1 2506.656,E2 2506.656} C_VEL
LIN {X 0,Y 720.177,Z 780.81,A -85,B 0,C 180,E1 2510.457,E2 2510.457} C_VEL
LIN {X 0,Y 720.102,Z 780.81,A -85,B 0,C 180,E1 2515.188,E2 2515.188} C_VEL
LIN {X 0,Y 720.179,Z 780.81,A -85,B 0,C 180,E1 2520.002,E2 2520.002} C_VEL
LIN {X 0,Y 720.363,Z 780.81,A -85,B 0,C 180,E1 2524.814,E2 2524.814} C_VEL
LIN {X 0,Y 720.143,Z 780.81,A -85,B 0,C 180,E1 2529.664,E2 2529.664} C_VEL
LIN {X 0,Y 720.026,Z 780.81,A -85,B 0,C 180,E1 2534.586,E2 2534.586} C_VEL
LIN {X 0,Y 720.051,Z 780.81,A -85,B 0,C 180,E1 2539.203,E2 2539.203} C_VEL
LIN {X 0,Y 719.971,Z 780.81,A -85,B 0,C 180,E1 2544.817,E2 2544.817} C_VEL
LIN {X 0,Y 719.918,Z 780.81,A -85,B 0,C 180,E1 2550.245,E2 2550.245} C_VEL
LIN {X 0,Y 719.842,Z 780.81,A -85,B 0,C 180,E1 2555.047,E2 2555.047} C_VEL
LIN {X 0,Y 719.673,Z 780.81,A -85,B 0,C 180,E1 2559.038,E2 2559.038} C_VEL
LIN {X 0,Y 720.02,Z 780.81,A -85,B 0,C 180,E1 2563.827,E2 2563.827} C_VEL
LIN {X 0,Y 719.828,Z 780.81,A -85,B 0,C 180,E1 2569.401,E2 2569.401} C_VEL
LIN {X 0,Y 719.947,Z 780.81,A -85,B 0,C 180,E1 2574.007,E2 2574.007} C_VEL
LIN {X 0,Y 719.931,Z 780.81,A -85,B 0,C 180,E1 2575.864,E2 2575.864} C_VEL
LIN {X 0,Y 726.15,Z 797.899,A -85,B 0,C 180,E1 2576.381,E2 2576.381} C_VEL
LIN {X 0,Y 725.704,Z 842.867,A -85,B 0,C 180,E1 2577.186,E2 2577.186} C_VEL
LIN {X 0,Y 724.887,Z 889.804,A -85,B 0,C 180,E1 2578.591,E2 2578.591} C_VEL
LIN {X 0,Y 723.926,Z 933.218,A -85,B 0,C 180,E1 2580.469,E2 2580.469} C_VEL
LIN {X 0,Y 722.93,Z 972.254,A -85,B 0,C 180,E1 2582.713,E2 2582.713} C_VEL
LIN {X 0,Y 722.063,Z 1006.907,A -85,B 0,C 180,E1 2585.258,E2 2585.258} C_VEL
LIN {X 0,Y 721.413,Z 1037.117,A -85,B 0,C 180,E1 2588.047,E2 2588.047} C_VEL
LIN {X 0,Y 720.823,Z 1065.451,A -85,B 0,C 180,E1 2591.394,E2 2591.394} C_VEL
LIN {X 0,Y 720.474,Z 1087.289,A -85,B 0,C 180,E1 2594.815,E2 2594.815} C_VEL
LIN {X 0,Y 720.327,Z 1102.924,A -85,B 0,C 180,E1 2598.198,E2 2598.198} C_VEL
LIN {X 0,Y 720.236,Z 1113.279,A -85,B 0,C 180,E1 2601.555,E2 2601.555} C_VEL
LIN {X 0,Y 720.187,Z 1118.761,A -85,B 0,C 180,E1 2605.186,E2 2605.186} C_VEL
LIN {X 0,Y 720.172,Z 1118.698,A -85,B 0,C 180,E1 2608.798,E2 2608.798} C_VEL
LIN {X 0,Y 720.221,Z 1113.148,A -85,B 0,C 180,E1 2612.406,E2 2612.406} C_VEL
LIN {X 0,Y 720.269,Z 1103.264,A -85,B 0,C 180,E1 2615.622,E2 2615.622} C_VEL
LIN {X 0,Y 720.428,Z 1089.187,A -85,B 0,C 180,E1 2618.748,E2 2618.748} C_VEL
LIN {X 0,Y 720.75,Z 1069.447,A -85,B 0,C 180,E1 2621.949,E2 2621.949} C_VEL
LIN {X 0,Y 721.167,Z 1044.845,A -85,B 0,C 180,E1 2625.035,E2 2625.035} C_VEL
LIN {X 0,Y 721.888,Z 1012.839,A -85,B 0,C 180,E1 2628.159,E2 2628.159} C_VEL
LIN {X 0,Y 722.843,Z 976.724,A -85,B 0,C 180,E1 2630.907,E2 2630.907} C_VEL
LIN {X 0,Y 723.893,Z 935.808,A -85,B 0,C 180,E1 2633.312,E2 2633.312} C_VEL
LIN {X 0,Y 724.843,Z 892.353,A -85,B 0,C 180,E1 2635.221,E2 2635.221} C_VEL
LIN {X 0,Y 725.606,Z 848.911,A -85,B 0,C 180,E1 2636.571,E2 2636.571} C_VEL
LIN {X 0,Y 726.216,Z 806.428,A -85,B 0,C 180,E1 2637.412,E2 2637.412} C_VEL
LIN {X 0,Y 724.784,Z 792.287,A -85,B 0,C 180,E1 2637.668,E2 2637.668} C_VEL
LIN {X 0,Y 720.233,Z 780.81,A -85,B 0,C 180,E1 2638.032,E2 2638.032} C_VEL
LIN {X 0,Y 720.028,Z 780.81,A -85,B 0,C 180,E1 2643.07,E2 2643.07} C_VEL
LIN {X 0,Y 719.87,Z 780.81,A -85,B 0,C 180,E1 2647.5,E2 2647.5} C_VEL
LIN {X 0,Y 719.963,Z 780.81,A -85,B 0,C 180,E1 2652.734,E2 2652.734} C_VEL
LIN {X 0,Y 719.696,Z 780.81,A -85,B 0,C 180,E1 2657.298,E2 2657.298} C_VEL
LIN {X 0,Y 719.773,Z 780.81,A -85,B 0,C 180,E1 2662.5,E2 2662.5} C_VEL
LIN {X 0,Y 719.825,Z 780.81,A -85,B 0,C 180,E1 2667.11,E2 2667.11} C_VEL
LIN {X 0,Y 719.928,Z 780.81,A -85,B 0,C 180,E1 2671.833,E2 2671.833} C_VEL
LIN {X 0,Y 719.97,Z 780.81,A -85,B 0,C 180,E1 2676.5,E2 2676.5} C_VEL
LIN {X 0,Y 720.082,Z 780.81,A -85,B 0,C 180,E1 2681.654,E2 2681.654} C_VEL
LIN {X 0,Y 720.001,Z 780.81,A -85,B 0,C 180,E1 2686.653,E2 2686.653} C_VEL
LIN {X 0,Y 720.207,Z 780.81,A -85,B 0,C 180,E1 2690.451,E2 2690.451} C_VEL
LIN {X 0,Y 720.119,Z 780.81,A -85,B 0,C 180,E1 2695.184,E2 2695.184} C_VEL
LIN {X 0,Y 720.217,Z 780.81,A -85,B 0,C 180,E1 2699.998,E2 2699.998} C_VEL
LIN {X 0,Y 720.325,Z 780.81,A -85,B 0,C 180,E1 2704.811,E2 2704.811} C_VEL
LIN {X 0,Y 720.148,Z 780.81,A -85,B 0,C 180,E1 2708.951,E2 2708.951} C_VEL
LIN {X 0,Y 716.112,Z 780.81,A -85,B 0,C 180,E1 2710.306,E2 2710.306} C_VEL
LIN {X 0,Y 712.151,Z 780.81,A -85,B 0,C 180,E1 2711.675,E2 2711.675} C_VEL
LIN {X 0,Y 712.249,Z 780.81,A -85,B 0,C 180,E1 2717.306,E2 2717.306} C_VEL
LIN {X 0,Y 712.07,Z 780.81,A -85,B 0,C 180,E1 2722.45,E2 2722.45} C_VEL
LIN {X 0,Y 712.022,Z 780.81,A -85,B 0,C 180,E1 2726.955,E2 2726.955} C_VEL
LIN {X 0,Y 712.11,Z 780.81,A -85,B 0,C 180,E1 2732.031,E2 2732.031} C_VEL
LIN {X 0,Y 712.006,Z 780.81,A -85,B 0,C 180,E1 2736.45,E2 2736.45} C_VEL
LIN {X 0,Y 711.885,Z 780.81,A -85,B 0,C 180,E1 2742.017,E2 2742.017} C_VEL
LIN {X 0,Y 711.949,Z 780.81,A -85,B 0,C 180,E1 2747.218,E2 2747.218} C_VEL
LIN {X 0,Y 711.873,Z 780.81,A -85,B 0,C 180,E1 2752.005,E2 2752.005} C_VEL
LIN {X 0,Y 712.061,Z 780.81,A -85,B 0,C 180,E1 2756.511,E2 2756.511} C_VEL
LIN {X 0,Y 712.184,Z 781.59,A -85,B 0,C 180,E1 2758.094,E2 2758.094} C_VEL
LIN {X 0,Y 719.322,Z 798.149,A -85,B 0,C 180,E1 2758.638,E2 2758.638} C_VEL
LIN {X 0,Y 719.169,Z 863.78,A -85,B 0,C 180,E1 2759.512,E2 2759.512} C_VEL
LIN {X 0,Y 718.42,Z 907.278,A -85,B 0,C 180,E1 2760.587,E2 2760.587} C_VEL
LIN {X 0,Y 717.371,Z 948.96,A -85,B 0,C 180,E1 2762.098,E2 2762.098} C_VEL
LIN {X 0,Y 716.211,Z 990.038,A -85,B 0,C 180,E1 2764.124,E2 2764.124} C_VEL
LIN {X 0,Y 715.042,Z 1029.466,A -85,B 0,C 180,E1 2766.686,E2 2766.686} C_VEL
LIN {X 0,Y 713.992,Z 1063.865,A -85,B 0,C 180,E1 2769.56,E2 2769.56} C_VEL
LIN {X 0,Y 713.243,Z 1093.632,A -85,B 0,C 180,E1 2772.745,E2 2772.745} C_VEL
LIN {X 0,Y 712.789,Z 1116.456,A -85,B 0,C 180,E1 2775.888,E2 2775.888} C_VEL
LIN {X 0,Y 712.462,Z 1135.27,A -85,B 0,C 180,E1 2779.304,E2 2779.304} C_VEL
LIN {X 0,Y 712.349,Z 1148.22,A -85,B 0,C 180,E1 2782.687,E2 2782.687} C_VEL
LIN {X 0,Y 712.443,Z 1154.868,A -85,B 0,C 180,E1 2785.327,E2 2785.327} C_VEL
LIN {X 0,Y 712.344,Z 1159.17,A -85,B 0,C 180,E1 2788.784,E2 2788.784} C_VEL
LIN {X 0,Y 712.299,Z 1158.226,A -85,B 0,C 180,E1 2792.431,E2 2792.431} C_VEL
LIN {X 0,Y 712.39,Z 1151.679,A -85,B 0,C 180,E1 2796.087,E2 2796.087} C_VEL
LIN {X 0,Y 712.437,Z 1140.769,A -85,B 0,C 180,E1 2799.429,E2 2799.429} C_VEL
LIN {X 0,Y 712.641,Z 1124.418,A -85,B 0,C 180,E1 2802.787,E2 2802.787} C_VEL
LIN {X 0,Y 713.013,Z 1103.533,A -85,B 0,C 180,E1 2805.992,E2 2805.992} C_VEL
LIN {X 0,Y 713.677,Z 1076.112,A -85,B 0,C 180,E1 2809.23,E2 2809.23} C_VEL
LIN {X 0,Y 714.664,Z 1041.721,A -85,B 0,C 180,E1 2812.37,E2 2812.37} C_VEL
LIN {X 0,Y 715.839,Z 1003.822,A -85,B 0,C 180,E1 2815.055,E2 2815.055} C_VEL
LIN {X 0,Y 717.038,Z 962.825,A -85,B 0,C 180,E1 2817.281,E2 2817.281} C_VEL
LIN {X 0,Y 718.095,Z 921.715,A -85,B 0,C 180,E1 2818.946,E2 2818.946} C_VEL
LIN {X 0,Y 718.977,Z 881.207,A -85,B 0,C 180,E1 2820.118,E2 2820.118} C_VEL
LIN {X 0,Y 719.508,Z 837.911,A -85,B 0,C 180,E1 2820.887,E2 2820.887} C_VEL
LIN {X 0,Y 718.552,Z 796.014,A -85,B 0,C 180,E1 2821.424,E2 2821.424} C_VEL
LIN {X 0,Y 712.248,Z 780.81,A -85,B 0,C 180,E1 2821.955,E2 2821.955} C_VEL
LIN {X 0,Y 711.975,Z 780.81,A -85,B 0,C 180,E1 2826.46,E2 2826.46} C_VEL
LIN {X 0,Y 712.06,Z 780.81,A -85,B 0,C 180,E1 2832.047,E2 2832.047} C_VEL
LIN {X 0,Y 711.968,Z 780.81,A -85,B 0,C 180,E1 2836.188,E2 2836.188} C_VEL
LIN {X 0,Y 711.943,Z 780.81,A -85,B 0,C 180,E1 2841.75,E2 2841.75} C_VEL
LIN {X 0,Y 711.873,Z 780.81,A -85,B 0,C 180,E1 2846.511,E2 2846.511} C_VEL
LIN {X 0,Y 711.977,Z 780.81,A -85,B 0,C 180,E1 2850.788,E2 2850.788} C_VEL
LIN {X 0,Y 712.096,Z 780.81,A -85,B 0,C 180,E1 2854.893,E2 2854.893} C_VEL
LIN {X 0,Y 712.07,Z 780.81,A -85,B 0,C 180,E1 2860.157,E2 2860.157} C_VEL
LIN {X 0,Y 712.171,Z 780.81,A -85,B 0,C 180,E1 2863.993,E2 2863.993} C_VEL
LIN {X 0,Y 712.273,Z 780.81,A -85,B 0,C 180,E1 2868.996,E2 2868.996} C_VEL
LIN {X 0,Y 712.308,Z 780.81,A -85,B 0,C 180,E1 2873.914,E2 2873.914} C_VEL
LIN {X 0,Y 712.213,Z 780.81,A -85,B 0,C 180,E1 2878.786,E2 2878.786} C_VEL
LIN {X 0,Y 712.214,Z 780.81,A -85,B 0,C 180,E1 2882.433,E2 2882.433} C_VEL
LIN {X 0,Y 712.248,Z 780.81,A -85,B 0,C 180,E1 2886.09,E2 2886.09} C_VEL
LIN {X 0,Y 712.159,Z 780.81,A -85,B 0,C 180,E1 2891.009,E2 2891.009} C_VEL
LIN {X 0,Y 712.238,Z 780.81,A -85,B 0,C 180,E1 2896.01,E2 2896.01} C_VEL
LIN {X 0,Y 712.089,Z 780.81,A -85,B 0,C 180,E1 2901.145,E2 2901.145} C_VEL
LIN {X 0,Y 711.979,Z 780.81,A -85,B 0,C 180,E1 2906.466,E2 2906.466} C_VEL
LIN {X 0,Y 712.067,Z 780.81,A -85,B 0,C 180,E1 2911.914,E2 2911.914} C_VEL
LIN {X 0,Y 711.993,Z 780.81,A -85,B 0,C 180,E1 2916.455,E2 2916.455} C_VEL
LIN {X 0,Y 712.07,Z 780.81,A -85,B 0,C 180,E1 2922.765,E2 2922.765} C_VEL
LIN {X 0,Y 711.824,Z 780.81,A -85,B 0,C 180,E1 2927.211,E2 2927.211} C_VEL
LIN {X 0,Y 712.086,Z 780.81,A -85,B 0,C 180,E1 2932.02,E2 2932.02} C_VEL
LIN {X 0,Y 712,Z 780.81,A -85,B 0,C 180,E1 2935.489,E2 2935.489} C_VEL
LIN {X 0,Y 719.34,Z 799.145,A -85,B 0,C 180,E1 2936.076,E2 2936.076} C_VEL
LIN {X 0,Y 718.782,Z 844.148,A -85,B 0,C 180,E1 2936.903,E2 2936.903} C_VEL
LIN {X 0,Y 717.809,Z 890.517,A -85,B 0,C 180,E1 2938.313,E2 2938.313} C_VEL
LIN {X 0,Y 716.653,Z 934.849,A -85,B 0,C 180,E1 2940.261,E2 2940.261} C_VEL
LIN {X 0,Y 715.421,Z 976.106,A -85,B 0,C 180,E1 2942.697,E2 2942.697} C_VEL
LIN {X 0,Y 714.333,Z 1013.188,A -85,B 0,C 180,E1 2945.546,E2 2945.546} C_VEL
LIN {X 0,Y 713.457,Z 1045.243,A -85,B 0,C 180,E1 2948.716,E2 2948.716} C_VEL
LIN {X 0,Y 712.855,Z 1071.115,A -85,B 0,C 180,E1 2952.03,E2 2952.03} C_VEL
LIN {X 0,Y 712.583,Z 1090.318,A -85,B 0,C 180,E1 2955.258,E2 2955.258} C_VEL
LIN {X 0,Y 712.467,Z 1105.112,A -85,B 0,C 180,E1 2958.687,E2 2958.687} C_VEL
LIN {X 0,Y 712.374,Z 1114.464,A -85,B 0,C 180,E1 2962.076,E2 2962.076} C_VEL
LIN {X 0,Y 712.294,Z 1119.057,A -85,B 0,C 180,E1 2965.523,E2 2965.523} C_VEL
LIN {X 0,Y 712.272,Z 1118.726,A -85,B 0,C 180,E1 2968.785,E2 2968.785} C_VEL
LIN {X 0,Y 712.326,Z 1113.235,A -85,B 0,C 180,E1 2972.432,E2 2972.432} C_VEL
LIN {X 0,Y 712.403,Z 1103.022,A -85,B 0,C 180,E1 2975.783,E2 2975.783} C_VEL
LIN {X 0,Y 712.573,Z 1087.84,A -85,B 0,C 180,E1 2979.133,E2 2979.133} C_VEL
LIN {X 0,Y 713.05,Z 1066.096,A -85,B 0,C 180,E1 2982.597,E2 2982.597} C_VEL
LIN {X 0,Y 713.614,Z 1039.404,A -85,B 0,C 180,E1 2985.828,E2 2985.828} C_VEL
LIN {X 0,Y 714.382,Z 1009.7,A -85,B 0,C 180,E1 2988.66,E2 2988.66} C_VEL
LIN {X 0,Y 715.472,Z 974.686,A -85,B 0,C 180,E1 2991.305,E2 2991.305} C_VEL
LIN {X 0,Y 716.659,Z 935.455,A -85,B 0,C 180,E1 2993.618,E2 2993.618} C_VEL
LIN {X 0,Y 717.787,Z 891.203,A -85,B 0,C 180,E1 2995.57,E2 2995.57} C_VEL
LIN {X 0,Y 718.761,Z 846.51,A -85,B 0,C 180,E1 2996.945,E2 2996.945} C_VEL
LIN {X 0,Y 719.381,Z 803.791,A -85,B 0,C 180,E1 2997.769,E2 2997.769} C_VEL
LIN {X 0,Y 717.673,Z 793.814,A -85,B 0,C 180,E1 2997.986,E2 2997.986} C_VEL
LIN {X 0,Y 712.206,Z 780.81,A -85,B 0,C 180,E1 2998.454,E2 2998.454} C_VEL
LIN {X 0,Y 712.037,Z 780.81,A -85,B 0,C 180,E1 3003.49,E2 3003.49} C_VEL
LIN {X 0,Y 711.816,Z 780.81,A -85,B 0,C 180,E1 3008.246,E2 3008.246} C_VEL
LIN {X 0,Y 712.127,Z 780.81,A -85,B 0,C 180,E1 3013.832,E2 3013.832} C_VEL
LIN {X 0,Y 711.821,Z 780.81,A -85,B 0,C 180,E1 3018.852,E2 3018.852} C_VEL
LIN {X 0,Y 711.908,Z 780.81,A -85,B 0,C 180,E1 3023.765,E2 3023.765} C_VEL
LIN {X 0,Y 712.002,Z 780.81,A -85,B 0,C 180,E1 3029.382,E2 3029.382} C_VEL
LIN {X 0,Y 712.157,Z 780.81,A -85,B 0,C 180,E1 3033.542,E2 3033.542} C_VEL
LIN {X 0,Y 712.091,Z 780.81,A -85,B 0,C 180,E1 3039.022,E2 3039.022} C_VEL
LIN {X 0,Y 712.191,Z 780.81,A -85,B 0,C 180,E1 3043.989,E2 3043.989} C_VEL
LIN {X 0,Y 712.299,Z 780.81,A -85,B 0,C 180,E1 3048.993,E2 3048.993} C_VEL
LIN {X 0,Y 712.346,Z 780.81,A -85,B 0,C 180,E1 3053.911,E2 3053.911} C_VEL
LIN {X 0,Y 712.249,Z 780.81,A -85,B 0,C 180,E1 3058.783,E2 3058.783} C_VEL
LIN {X 0,Y 712.206,Z 780.81,A -85,B 0,C 180,E1 3062.43,E2 3062.43} C_VEL
LIN {X 0,Y 712.213,Z 780.81,A -85,B 0,C 180,E1 3066.087,E2 3066.087} C_VEL
LIN {X 0,Y 712.155,Z 780.81,A -85,B 0,C 180,E1 3071.006,E2 3071.006} C_VEL
LIN {X 0,Y 712.151,Z 780.81,A -85,B 0,C 180,E1 3071.675,E2 3071.675} C_VEL
LIN {X 0,Y 710.921,Z 780.81,A -85,B 0,C 180,E1 3072.371,E2 3072.371} C_VEL
LIN {X 0,Y 704.297,Z 780.81,A -85,B 0,C 180,E1 3074.259,E2 3074.259} C_VEL
LIN {X 0,Y 704.204,Z 780.81,A -85,B 0,C 180,E1 3074.437,E2 3074.437} C_VEL
LIN {X 0,Y 704.258,Z 780.81,A -85,B 0,C 180,E1 3079.247,E2 3079.247} C_VEL
LIN {X 0,Y 704.205,Z 780.81,A -85,B 0,C 180,E1 3084.054,E2 3084.054} C_VEL
LIN {X 0,Y 704.11,Z 780.81,A -85,B 0,C 180,E1 3089.57,E2 3089.57} C_VEL
LIN {X 0,Y 704.129,Z 780.81,A -85,B 0,C 180,E1 3093.907,E2 3093.907} C_VEL
LIN {X 0,Y 703.912,Z 780.81,A -85,B 0,C 180,E1 3098.492,E2 3098.492} C_VEL
LIN {X 0,Y 703.985,Z 780.81,A -85,B 0,C 180,E1 3103.372,E2 3103.372} C_VEL
LIN {X 0,Y 703.973,Z 780.81,A -85,B 0,C 180,E1 3108.688,E2 3108.688} C_VEL
LIN {X 0,Y 704.021,Z 780.81,A -85,B 0,C 180,E1 3113.058,E2 3113.058} C_VEL
LIN {X 0,Y 704.216,Z 781.308,A -85,B 0,C 180,E1 3117.687,E2 3117.687} C_VEL
LIN {X 0,Y 712.622,Z 802.016,A -85,B 0,C 180,E1 3118.354,E2 3118.354} C_VEL
LIN {X 0,Y 712.335,Z 863.781,A -85,B 0,C 180,E1 3119.187,E2 3119.187} C_VEL
LIN {X 0,Y 711.461,Z 907.488,A -85,B 0,C 180,E1 3120.277,E2 3120.277} C_VEL
LIN {X 0,Y 710.262,Z 948.709,A -85,B 0,C 180,E1 3121.782,E2 3121.782} C_VEL
LIN {X 0,Y 708.937,Z 990.712,A -85,B 0,C 180,E1 3123.879,E2 3123.879} C_VEL
LIN {X 0,Y 707.545,Z 1029.715,A -85,B 0,C 180,E1 3126.442,E2 3126.442} C_VEL
LIN {X 0,Y 706.326,Z 1065.597,A -85,B 0,C 180,E1 3129.492,E2 3129.492} C_VEL
LIN {X 0,Y 705.419,Z 1096.262,A -85,B 0,C 180,E1 3132.869,E2 3132.869} C_VEL
LIN {X 0,Y 704.903,Z 1120.369,A -85,B 0,C 180,E1 3136.36,E2 3136.36} C_VEL
LIN {X 0,Y 704.56,Z 1137.955,A -85,B 0,C 180,E1 3139.808,E2 3139.808} C_VEL
LIN {X 0,Y 704.469,Z 1150.116,A -85,B 0,C 180,E1 3143.224,E2 3143.224} C_VEL
LIN {X 0,Y 704.423,Z 1156.666,A -85,B 0,C 180,E1 3146.309,E2 3146.309} C_VEL
LIN {X 0,Y 704.404,Z 1159.5,A -85,B 0,C 180,E1 3149.999,E2 3149.999} C_VEL
LIN {X 0,Y 704.379,Z 1156.668,A -85,B 0,C 180,E1 3153.689,E2 3153.689} C_VEL
LIN {X 0,Y 704.518,Z 1150.12,A -85,B 0,C 180,E1 3156.774,E2 3156.774} C_VEL
LIN {X 0,Y 704.565,Z 1137.961,A -85,B 0,C 180,E1 3160.191,E2 3160.191} C_VEL
LIN {X 0,Y 704.896,Z 1120.377,A -85,B 0,C 180,E1 3163.639,E2 3163.639} C_VEL
LIN {X 0,Y 705.476,Z 1096.273,A -85,B 0,C 180,E1 3167.128,E2 3167.128} C_VEL
LIN {X 0,Y 706.408,Z 1065.613,A -85,B 0,C 180,E1 3170.504,E2 3170.504} C_VEL
LIN {X 0,Y 707.61,Z 1029.643,A -85,B 0,C 180,E1 3173.561,E2 3173.561} C_VEL
LIN {X 0,Y 708.887,Z 989.881,A -85,B 0,C 180,E1 3176.172,E2 3176.172} C_VEL
LIN {X 0,Y 710.335,Z 947.219,A -85,B 0,C 180,E1 3178.282,E2 3178.282} C_VEL
LIN {X 0,Y 711.456,Z 904.153,A -85,B 0,C 180,E1 3179.828,E2 3179.828} C_VEL
LIN {X 0,Y 712.329,Z 861.23,A -85,B 0,C 180,E1 3180.859,E2 3180.859} C_VEL
LIN {X 0,Y 712.037,Z 798.883,A -85,B 0,C 180,E1 3181.712,E2 3181.712} C_VEL
LIN {X 0,Y 704.247,Z 780.81,A -85,B 0,C 180,E1 3182.351,E2 3182.351} C_VEL
LIN {X 0,Y 703.966,Z 780.81,A -85,B 0,C 180,E1 3187.434,E2 3187.434} C_VEL
LIN {X 0,Y 704.271,Z 780.81,A -85,B 0,C 180,E1 3193.361,E2 3193.361} C_VEL
LIN {X 0,Y 703.967,Z 780.81,A -85,B 0,C 180,E1 3198.702,E2 3198.702} C_VEL
LIN {X 0,Y 703.989,Z 780.81,A -85,B 0,C 180,E1 3203.067,E2 3203.067} C_VEL
LIN {X 0,Y 703.963,Z 780.81,A -85,B 0,C 180,E1 3207.553,E2 3207.553} C_VEL
LIN {X 0,Y 704.105,Z 780.81,A -85,B 0,C 180,E1 3211.833,E2 3211.833} C_VEL
LIN {X 0,Y 704.153,Z 780.81,A -85,B 0,C 180,E1 3215.944,E2 3215.944} C_VEL
LIN {X 0,Y 704.223,Z 780.81,A -85,B 0,C 180,E1 3221.23,E2 3221.23} C_VEL
LIN {X 0,Y 704.188,Z 780.81,A -85,B 0,C 180,E1 3226.351,E2 3226.351} C_VEL
LIN {X 0,Y 704.245,Z 780.81,A -85,B 0,C 180,E1 3231.365,E2 3231.365} C_VEL
LIN {X 0,Y 704.411,Z 780.81,A -85,B 0,C 180,E1 3236.313,E2 3236.313} C_VEL
LIN {X 0,Y 704.549,Z 780.81,A -85,B 0,C 180,E1 3241.231,E2 3241.231} C_VEL
LIN {X 0,Y 704.338,Z 780.81,A -85,B 0,C 180,E1 3246.159,E2 3246.159} C_VEL
LIN {X 0,Y 704.251,Z 780.81,A -85,B 0,C 180,E1 3251.134,E2 3251.134} C_VEL
LIN {X 0,Y 704.316,Z 780.81,A -85,B 0,C 180,E1 3256.194,E2 3256.194} C_VEL
LIN {X 0,Y 704.15,Z 780.81,A -85,B 0,C 180,E1 3261.395,E2 3261.395} C_VEL
LIN {X 0,Y 704.094,Z 780.81,A -85,B 0,C 180,E1 3265.66,E2 3265.66} C_VEL
LIN {X 0,Y 704.093,Z 780.81,A -85,B 0,C 180,E1 3270.999,E2 3270.999} C_VEL
LIN {X 0,Y 704.037,Z 780.81,A -85,B 0,C 180,E1 3275.412,E2 3275.412} C_VEL
LIN {X 0,Y 703.834,Z 780.81,A -85,B 0,C 180,E1 3280.092,E2 3280.092} C_VEL
LIN {X 0,Y 704.149,Z 780.81,A -85,B 0,C 180,E1 3285.08,E2 3285.08} C_VEL
LIN {X 0,Y 704.106,Z 780.81,A -85,B 0,C 180,E1 3290.58,E2 3290.58} C_VEL
LIN {X 0,Y 704.102,Z 780.984,A -85,B 0,C 180,E1 3295.104,E2 3295.104} C_VEL
LIN {X 0,Y 712.584,Z 801.55,A -85,B 0,C 180,E1 3295.784,E2 3295.784} C_VEL
LIN {X 0,Y 711.871,Z 845.736,A -85,B 0,C 180,E1 3296.624,E2 3296.624} C_VEL
LIN {X 0,Y 710.807,Z 889.696,A -85,B 0,C 180,E1 3297.973,E2 3297.973} C_VEL
LIN {X 0,Y 709.454,Z 933.902,A -85,B 0,C 180,E1 3299.92,E2 3299.92} C_VEL
LIN {X 0,Y 708.065,Z 974.281,A -85,B 0,C 180,E1 3302.306,E2 3302.306} C_VEL
LIN {X 0,Y 706.856,Z 1009.375,A -85,B 0,C 180,E1 3304.979,E2 3304.979} C_VEL
LIN {X 0,Y 705.984,Z 1039.108,A -85,B 0,C 180,E1 3307.837,E2 3307.837} C_VEL
LIN {X 0,Y 705.33,Z 1065.546,A -85,B 0,C 180,E1 3311.056,E2 3311.056} C_VEL
LIN {X 0,Y 704.805,Z 1087.644,A -85,B 0,C 180,E1 3314.606,E2 3314.606} C_VEL
LIN {X 0,Y 704.562,Z 1102.664,A -85,B 0,C 180,E1 3317.93,E2 3317.93} C_VEL
LIN {X 0,Y 704.453,Z 1113.105,A -85,B 0,C 180,E1 3321.365,E2 3321.365} C_VEL
LIN {X 0,Y 704.414,Z 1118.705,A -85,B 0,C 180,E1 3325.078,E2 3325.078} C_VEL
LIN {X 0,Y 704.372,Z 1118.755,A -85,B 0,C 180,E1 3328.771,E2 3328.771} C_VEL
LIN {X 0,Y 704.447,Z 1113.322,A -85,B 0,C 180,E1 3332.46,E2 3332.46} C_VEL
LIN {X 0,Y 704.521,Z 1103.15,A -85,B 0,C 180,E1 3335.848,E2 3335.848} C_VEL
LIN {X 0,Y 704.715,Z 1088.774,A -85,B 0,C 180,E1 3339.098,E2 3339.098} C_VEL
LIN {X 0,Y 705.213,Z 1067.854,A -85,B 0,C 180,E1 3342.52,E2 3342.52} C_VEL
LIN {X 0,Y 705.822,Z 1042.736,A -85,B 0,C 180,E1 3345.676,E2 3345.676} C_VEL
LIN {X 0,Y 706.752,Z 1012.01,A -85,B 0,C 180,E1 3348.707,E2 3348.707} C_VEL
LIN {X 0,Y 708.007,Z 977.206,A -85,B 0,C 180,E1 3351.409,E2 3351.409} C_VEL
LIN {X 0,Y 709.407,Z 936.155,A -85,B 0,C 180,E1 3353.874,E2 3353.874} C_VEL
LIN {X 0,Y 710.708,Z 892.202,A -85,B 0,C 180,E1 3355.841,E2 3355.841} C_VEL
LIN {X 0,Y 711.819,Z 848.273,A -85,B 0,C 180,E1 3357.221,E2 3357.221} C_VEL
LIN {X 0,Y 712.574,Z 804.26,A -85,B 0,C 180,E1 3358.089,E2 3358.089} C_VEL
LIN {X 0,Y 710.86,Z 796.461,A -85,B 0,C 180,E1 3358.28,E2 3358.28} C_VEL
LIN {X 0,Y 704.219,Z 780.81,A -85,B 0,C 180,E1 3358.874,E2 3358.874} C_VEL
LIN {X 0,Y 704.103,Z 780.81,A -85,B 0,C 180,E1 3363.918,E2 3363.918} C_VEL
LIN {X 0,Y 703.888,Z 780.81,A -85,B 0,C 180,E1 3368.505,E2 3368.505} C_VEL
LIN {X 0,Y 704.186,Z 780.81,A -85,B 0,C 180,E1 3373.369,E2 3373.369} C_VEL
LIN {X 0,Y 703.925,Z 780.81,A -85,B 0,C 180,E1 3378.708,E2 3378.708} C_VEL
LIN {X 0,Y 703.928,Z 780.81,A -85,B 0,C 180,E1 3383.059,E2 3383.059} C_VEL
LIN {X 0,Y 703.974,Z 780.81,A -85,B 0,C 180,E1 3387.549,E2 3387.549} C_VEL
LIN {X 0,Y 704.11,Z 780.81,A -85,B 0,C 180,E1 3391.829,E2 3391.829} C_VEL
LIN {X 0,Y 704.148,Z 780.81,A -85,B 0,C 180,E1 3395.939,E2 3395.939} C_VEL
LIN {X 0,Y 704.235,Z 780.81,A -85,B 0,C 180,E1 3401.226,E2 3401.226} C_VEL
LIN {X 0,Y 704.211,Z 780.81,A -85,B 0,C 180,E1 3406.348,E2 3406.348} C_VEL
LIN {X 0,Y 704.29,Z 780.81,A -85,B 0,C 180,E1 3411.362,E2 3411.362} C_VEL
LIN {X 0,Y 704.436,Z 780.81,A -85,B 0,C 180,E1 3416.309,E2 3416.309} C_VEL
LIN {X 0,Y 704.576,Z 780.81,A -85,B 0,C 180,E1 3421.227,E2 3421.227} C_VEL
LIN {X 0,Y 704.304,Z 780.81,A -85,B 0,C 180,E1 3426.155,E2 3426.155} C_VEL
LIN {X 0,Y 704.248,Z 780.81,A -85,B 0,C 180,E1 3431.131,E2 3431.131} C_VEL
LIN {X 0,Y 704.204,Z 780.81,A -85,B 0,C 180,E1 3434.437,E2 3434.437} C_VEL
LIN {X 0,Y 700.275,Z 780.81,A -85,B 0,C 180,E1 3435.828,E2 3435.828} C_VEL
LIN {X 0,Y 696.412,Z 780.81,A -85,B 0,C 180,E1 3437.234,E2 3437.234} C_VEL
LIN {X 0,Y 696.274,Z 780.81,A -85,B 0,C 180,E1 3441.645,E2 3441.645} C_VEL
LIN {X 0,Y 696.27,Z 780.81,A -85,B 0,C 180,E1 3445.718,E2 3445.718} C_VEL
LIN {X 0,Y 696.185,Z 780.81,A -85,B 0,C 180,E1 3449.941,E2 3449.941} C_VEL
LIN {X 0,Y 696.163,Z 780.81,A -85,B 0,C 180,E1 3454.427,E2 3454.427} C_VEL
LIN {X 0,Y 695.964,Z 780.81,A -85,B 0,C 180,E1 3459.015,E2 3459.015} C_VEL
LIN {X 0,Y 695.985,Z 780.81,A -85,B 0,C 180,E1 3464.234,E2 3464.234} C_VEL
LIN {X 0,Y 695.965,Z 780.81,A -85,B 0,C 180,E1 3469.444,E2 3469.444} C_VEL
LIN {X 0,Y 696.13,Z 780.81,A -85,B 0,C 180,E1 3474.119,E2 3474.119} C_VEL
LIN {X 0,Y 696.264,Z 780.908,A -85,B 0,C 180,E1 3477.267,E2 3477.267} C_VEL
LIN {X 0,Y 705.927,Z 804.535,A -85,B 0,C 180,E1 3478.048,E2 3478.048} C_VEL
LIN {X 0,Y 705.514,Z 865.725,A -85,B 0,C 180,E1 3478.894,E2 3478.894} C_VEL
LIN {X 0,Y 704.494,Z 909.589,A -85,B 0,C 180,E1 3480.02,E2 3480.02} C_VEL
LIN {X 0,Y 703.15,Z 949.849,A -85,B 0,C 180,E1 3481.524,E2 3481.524} C_VEL
LIN {X 0,Y 701.622,Z 991.377,A -85,B 0,C 180,E1 3483.627,E2 3483.627} C_VEL
LIN {X 0,Y 700.045,Z 1030.855,A -85,B 0,C 180,E1 3486.263,E2 3486.263} C_VEL
LIN {X 0,Y 698.684,Z 1065.598,A -85,B 0,C 180,E1 3489.258,E2 3489.258} C_VEL
LIN {X 0,Y 697.668,Z 1096.263,A -85,B 0,C 180,E1 3492.673,E2 3492.673} C_VEL
LIN {X 0,Y 697.061,Z 1120.368,A -85,B 0,C 180,E1 3496.204,E2 3496.204} C_VEL
LIN {X 0,Y 696.68,Z 1137.955,A -85,B 0,C 180,E1 3499.691,E2 3499.691} C_VEL
LIN {X 0,Y 696.589,Z 1150.116,A -85,B 0,C 180,E1 3503.147,E2 3503.147} C_VEL
LIN {X 0,Y 696.544,Z 1156.665,A -85,B 0,C 180,E1 3506.268,E2 3506.268} C_VEL
LIN {X 0,Y 696.505,Z 1159.5,A -85,B 0,C 180,E1 3509.999,E2 3509.999} C_VEL
LIN {X 0,Y 696.492,Z 1156.581,A -85,B 0,C 180,E1 3513.794,E2 3513.794} C_VEL
LIN {X 0,Y 696.644,Z 1150.12,A -85,B 0,C 180,E1 3516.851,E2 3516.851} C_VEL
LIN {X 0,Y 696.695,Z 1137.962,A -85,B 0,C 180,E1 3520.307,E2 3520.307} C_VEL
LIN {X 0,Y 697.075,Z 1120.375,A -85,B 0,C 180,E1 3523.795,E2 3523.795} C_VEL
LIN {X 0,Y 697.735,Z 1096.274,A -85,B 0,C 180,E1 3527.324,E2 3527.324} C_VEL
LIN {X 0,Y 698.779,Z 1065.613,A -85,B 0,C 180,E1 3530.738,E2 3530.738} C_VEL
LIN {X 0,Y 700.122,Z 1029.764,A -85,B 0,C 180,E1 3533.819,E2 3533.819} C_VEL
LIN {X 0,Y 701.594,Z 990.416,A -85,B 0,C 180,E1 3536.433,E2 3536.433} C_VEL
LIN {X 0,Y 703.228,Z 948.066,A -85,B 0,C 180,E1 3538.555,E2 3538.555} C_VEL
LIN {X 0,Y 704.528,Z 904.634,A -85,B 0,C 180,E1 3540.136,E2 3540.136} C_VEL
LIN {X 0,Y 705.558,Z 860.769,A -85,B 0,C 180,E1 3541.196,E2 3541.196} C_VEL
LIN {X 0,Y 705.477,Z 801.803,A -85,B 0,C 180,E1 3542.007,E2 3542.007} C_VEL
LIN {X 0,Y 696.293,Z 780.81,A -85,B 0,C 180,E1 3542.771,E2 3542.771} C_VEL
LIN {X 0,Y 696.074,Z 780.81,A -85,B 0,C 180,E1 3547.433,E2 3547.433} C_VEL
LIN {X 0,Y 696.223,Z 780.81,A -85,B 0,C 180,E1 3552.457,E2 3552.457} C_VEL
LIN {X 0,Y 696.017,Z 780.81,A -85,B 0,C 180,E1 3557.71,E2 3557.71} C_VEL
LIN {X 0,Y 696.096,Z 780.81,A -85,B 0,C 180,E1 3562.577,E2 3562.577} C_VEL
LIN {X 0,Y 696.046,Z 780.81,A -85,B 0,C 180,E1 3567.851,E2 3567.851} C_VEL
LIN {X 0,Y 696.279,Z 780.81,A -85,B 0,C 180,E1 3572.894,E2 3572.894} C_VEL
LIN {X 0,Y 696.271,Z 780.81,A -85,B 0,C 180,E1 3578.355,E2 3578.355} C_VEL
LIN {X 0,Y 696.343,Z 780.81,A -85,B 0,C 180,E1 3583.619,E2 3583.619} C_VEL
LIN {X 0,Y 696.399,Z 780.81,A -85,B 0,C 180,E1 3588.742,E2 3588.742} C_VEL
LIN {X 0,Y 696.505,Z 780.81,A -85,B 0,C 180,E1 3593.775,E2 3593.775} C_VEL
LIN {X 0,Y 696.421,Z 780.81,A -85,B 0,C 180,E1 3598.759,E2 3598.759} C_VEL
LIN {X 0,Y 696.437,Z 780.81,A -85,B 0,C 180,E1 3602.489,E2 3602.489} C_VEL
LIN {X 0,Y 696.427,Z 780.81,A -85,B 0,C 180,E1 3606.229,E2 3606.229} C_VEL
LIN {X 0,Y 696.344,Z 780.81,A -85,B 0,C 180,E1 3611.263,E2 3611.263} C_VEL
LIN {X 0,Y 696.394,Z 780.81,A -85,B 0,C 180,E1 3616.384,E2 3616.384} C_VEL
LIN {X 0,Y 696.231,Z 780.81,A -85,B 0,C 180,E1 3621.65,E2 3621.65} C_VEL
LIN {X 0,Y 696.194,Z 780.81,A -85,B 0,C 180,E1 3625.726,E2 3625.726} C_VEL
LIN {X 0,Y 696.164,Z 780.81,A -85,B 0,C 180,E1 3629.946,E2 3629.946} C_VEL
LIN {X 0,Y 696.139,Z 780.81,A -85,B 0,C 180,E1 3634.427,E2 3634.427} C_VEL
LIN {X 0,Y 695.945,Z 780.81,A -85,B 0,C 180,E1 3639.021,E2 3639.021} C_VEL
LIN {X 0,Y 696.207,Z 780.81,A -85,B 0,C 180,E1 3644.255,E2 3644.255} C_VEL
LIN {X 0,Y 696.086,Z 780.81,A -85,B 0,C 180,E1 3649.438,E2 3649.438} C_VEL
LIN {X 0,Y 696.17,Z 780.81,A -85,B 0,C 180,E1 3654.476,E2 3654.476} C_VEL
LIN {X 0,Y 696.186,Z 780.86,A -85,B 0,C 180,E1 3654.696,E2 3654.696} C_VEL
LIN {X 0,Y 705.867,Z 804.241,A -85,B 0,C 180,E1 3655.491,E2 3655.491} C_VEL
LIN {X 0,Y 704.977,Z 847.943,A -85,B 0,C 180,E1 3656.355,E2 3656.355} C_VEL
LIN {X 0,Y 703.743,Z 891.55,A -85,B 0,C 180,E1 3657.729,E2 3657.729} C_VEL
LIN {X 0,Y 702.235,Z 934.913,A -85,B 0,C 180,E1 3659.671,E2 3659.671} C_VEL
LIN {X 0,Y 700.628,Z 976.078,A -85,B 0,C 180,E1 3662.149,E2 3662.149} C_VEL
LIN {X 0,Y 699.186,Z 1012.978,A -85,B 0,C 180,E1 3665.04,E2 3665.04} C_VEL
LIN {X 0,Y 698.083,Z 1044.727,A -85,B 0,C 180,E1 3668.242,E2 3668.242} C_VEL
LIN {X 0,Y 697.289,Z 1069.99,A -85,B 0,C 180,E1 3671.523,E2 3671.523} C_VEL
LIN {X 0,Y 696.877,Z 1089.968,A -85,B 0,C 180,E1 3674.918,E2 3674.918} C_VEL
LIN {X 0,Y 696.676,Z 1104.852,A -85,B 0,C 180,E1 3678.427,E2 3678.427} C_VEL
LIN {X 0,Y 696.583,Z 1114.33,A -85,B 0,C 180,E1 3681.895,E2 3681.895} C_VEL
LIN {X 0,Y 696.512,Z 1118.677,A -85,B 0,C 180,E1 3685.022,E2 3685.022} C_VEL
LIN {X 0,Y 696.472,Z 1118.783,A -85,B 0,C 180,E1 3688.757,E2 3688.757} C_VEL
LIN {X 0,Y 696.552,Z 1113.404,A -85,B 0,C 180,E1 3692.487,E2 3692.487} C_VEL
LIN {X 0,Y 696.632,Z 1103.278,A -85,B 0,C 180,E1 3695.915,E2 3695.915} C_VEL
LIN {X 0,Y 696.921,Z 1088.351,A -85,B 0,C 180,E1 3699.317,E2 3699.317} C_VEL
LIN {X 0,Y 697.539,Z 1065.713,A -85,B 0,C 180,E1 3703.011,E2 3703.011} C_VEL
LIN {X 0,Y 698.366,Z 1037.232,A -85,B 0,C 180,E1 3706.5,E2 3706.5} C_VEL
LIN {X 0,Y 699.49,Z 1004.365,A -85,B 0,C 180,E1 3709.612,E2 3709.612} C_VEL
LIN {X 0,Y 700.953,Z 968.652,A -85,B 0,C 180,E1 3712.254,E2 3712.254} C_VEL
LIN {X 0,Y 702.416,Z 930.387,A -85,B 0,C 180,E1 3714.465,E2 3714.465} C_VEL
LIN {X 0,Y 703.832,Z 887.685,A -85,B 0,C 180,E1 3716.327,E2 3716.327} C_VEL
LIN {X 0,Y 705.154,Z 841.357,A -85,B 0,C 180,E1 3717.723,E2 3717.723} C_VEL
LIN {X 0,Y 705.333,Z 801.63,A -85,B 0,C 180,E1 3718.482,E2 3718.482} C_VEL
LIN {X 0,Y 696.241,Z 780.81,A -85,B 0,C 180,E1 3719.281,E2 3719.281} C_VEL
LIN {X 0,Y 696.127,Z 780.81,A -85,B 0,C 180,E1 3724.435,E2 3724.435} C_VEL
LIN {X 0,Y 695.948,Z 780.81,A -85,B 0,C 180,E1 3729.027,E2 3729.027} C_VEL
LIN {X 0,Y 696.214,Z 780.81,A -85,B 0,C 180,E1 3734.262,E2 3734.262} C_VEL
LIN {X 0,Y 696.027,Z 780.81,A -85,B 0,C 180,E1 3739.453,E2 3739.453} C_VEL
LIN {X 0,Y 696.019,Z 780.81,A -85,B 0,C 180,E1 3744.118,E2 3744.118} C_VEL
LIN {X 0,Y 696.094,Z 780.81,A -85,B 0,C 180,E1 3748.604,E2 3748.604} C_VEL
LIN {X 0,Y 696.286,Z 780.81,A -85,B 0,C 180,E1 3752.89,E2 3752.89} C_VEL
LIN {X 0,Y 696.26,Z 780.81,A -85,B 0,C 180,E1 3758.351,E2 3758.351} C_VEL
LIN {X 0,Y 696.355,Z 780.81,A -85,B 0,C 180,E1 3763.615,E2 3763.615} C_VEL
LIN {X 0,Y 696.425,Z 780.81,A -85,B 0,C 180,E1 3768.739,E2 3768.739} C_VEL
LIN {X 0,Y 696.542,Z 780.81,A -85,B 0,C 180,E1 3773.772,E2 3773.772} C_VEL
LIN {X 0,Y 696.455,Z 780.81,A -85,B 0,C 180,E1 3778.755,E2 3778.755} C_VEL
LIN {X 0,Y 696.43,Z 780.81,A -85,B 0,C 180,E1 3782.485,E2 3782.485} C_VEL
LIN {X 0,Y 696.395,Z 780.81,A -85,B 0,C 180,E1 3786.226,E2 3786.226} C_VEL
LIN {X 0,Y 696.343,Z 780.81,A -85,B 0,C 180,E1 3791.259,E2 3791.259} C_VEL
LIN {X 0,Y 696.397,Z 780.81,A -85,B 0,C 180,E1 3796.38,E2 3796.38} C_VEL
LIN {X 0,Y 696.412,Z 780.81,A -85,B 0,C 180,E1 3797.234,E2 3797.234} C_VEL
LIN {X 0,Y 693.898,Z 780.81,A -85,B 0,C 180,E1 3798.292,E2 3798.292} C_VEL
LIN {X 0,Y 688.469,Z 780.81,A -85,B 0,C 180,E1 3799.873,E2 3799.873} C_VEL
LIN {X 0,Y 688.379,Z 780.81,A -85,B 0,C 180,E1 3800.056,E2 3800.056} C_VEL
LIN {X 0,Y 688.348,Z 780.81,A -85,B 0,C 180,E1 3804.645,E2 3804.645} C_VEL
LIN {X 0,Y 688.296,Z 780.81,A -85,B 0,C 180,E1 3808.874,E2 3808.874} C_VEL
LIN {X 0,Y 688.262,Z 780.81,A -85,B 0,C 180,E1 3813.455,E2 3813.455} C_VEL
LIN {X 0,Y 688.148,Z 780.81,A -85,B 0,C 180,E1 3817.931,E2 3817.931} C_VEL
LIN {X 0,Y 688.074,Z 780.81,A -85,B 0,C 180,E1 3823.553,E2 3823.553} C_VEL
LIN {X 0,Y 688.035,Z 780.81,A -85,B 0,C 180,E1 3828.785,E2 3828.785} C_VEL
LIN {X 0,Y 688.212,Z 780.81,A -85,B 0,C 180,E1 3834.315,E2 3834.315} C_VEL
LIN {X 0,Y 688.323,Z 781.084,A -85,B 0,C 180,E1 3836.843,E2 3836.843} C_VEL
LIN {X 0,Y 699.235,Z 807.207,A -85,B 0,C 180,E1 3837.737,E2 3837.737} C_VEL
LIN {X 0,Y 698.703,Z 866.407,A -85,B 0,C 180,E1 3838.572,E2 3838.572} C_VEL
LIN {X 0,Y 697.58,Z 909.705,A -85,B 0,C 180,E1 3839.695,E2 3839.695} C_VEL
LIN {X 0,Y 696.055,Z 949.795,A -85,B 0,C 180,E1 3841.204,E2 3841.204} C_VEL
LIN {X 0,Y 694.442,Z 990.411,A -85,B 0,C 180,E1 3843.273,E2 3843.273} C_VEL
LIN {X 0,Y 692.674,Z 1029.791,A -85,B 0,C 180,E1 3845.91,E2 3845.91} C_VEL
LIN {X 0,Y 691.07,Z 1065.598,A -85,B 0,C 180,E1 3849.018,E2 3849.018} C_VEL
LIN {X 0,Y 689.975,Z 1095.142,A -85,B 0,C 180,E1 3852.333,E2 3852.333} C_VEL
LIN {X 0,Y 689.289,Z 1118.422,A -85,B 0,C 180,E1 3855.721,E2 3855.721} C_VEL
LIN {X 0,Y 688.884,Z 1135.271,A -85,B 0,C 180,E1 3858.933,E2 3858.933} C_VEL
LIN {X 0,Y 688.687,Z 1148.22,A -85,B 0,C 180,E1 3862.434,E2 3862.434} C_VEL
LIN {X 0,Y 688.687,Z 1155.685,A -85,B 0,C 180,E1 3865.595,E2 3865.595} C_VEL
LIN {X 0,Y 688.67,Z 1159.169,A -85,B 0,C 180,E1 3868.742,E2 3868.742} C_VEL
LIN {X 0,Y 688.624,Z 1158.224,A -85,B 0,C 180,E1 3872.515,E2 3872.515} C_VEL
LIN {X 0,Y 688.781,Z 1153.236,A -85,B 0,C 180,E1 3875.665,E2 3875.665} C_VEL
LIN {X 0,Y 688.819,Z 1142.595,A -85,B 0,C 180,E1 3879.252,E2 3879.252} C_VEL
LIN {X 0,Y 689.101,Z 1127.474,A -85,B 0,C 180,E1 3882.666,E2 3882.666} C_VEL
LIN {X 0,Y 689.611,Z 1105.756,A -85,B 0,C 180,E1 3886.24,E2 3886.24} C_VEL
LIN {X 0,Y 690.512,Z 1079.696,A -85,B 0,C 180,E1 3889.497,E2 3889.497} C_VEL
LIN {X 0,Y 691.808,Z 1049.451,A -85,B 0,C 180,E1 3892.472,E2 3892.472} C_VEL
LIN {X 0,Y 693.344,Z 1014.985,A -85,B 0,C 180,E1 3895.16,E2 3895.16} C_VEL
LIN {X 0,Y 695.055,Z 975.806,A -85,B 0,C 180,E1 3897.542,E2 3897.542} C_VEL
LIN {X 0,Y 696.771,Z 933.47,A -85,B 0,C 180,E1 3899.468,E2 3899.468} C_VEL
LIN {X 0,Y 698.124,Z 891.275,A -85,B 0,C 180,E1 3900.841,E2 3900.841} C_VEL
LIN {X 0,Y 699.096,Z 848.328,A -85,B 0,C 180,E1 3901.746,E2 3901.746} C_VEL
LIN {X 0,Y 698.511,Z 803.732,A -85,B 0,C 180,E1 3902.342,E2 3902.342} C_VEL
LIN {X 0,Y 688.292,Z 780.81,A -85,B 0,C 180,E1 3903.198,E2 3903.198} C_VEL
LIN {X 0,Y 688.137,Z 780.81,A -85,B 0,C 180,E1 3907.941,E2 3907.941} C_VEL
LIN {X 0,Y 688.33,Z 780.81,A -85,B 0,C 180,E1 3913.59,E2 3913.59} C_VEL
LIN {X 0,Y 688.089,Z 780.81,A -85,B 0,C 180,E1 3918.801,E2 3918.801} C_VEL
LIN {X 0,Y 688.167,Z 780.81,A -85,B 0,C 180,E1 3923.648,E2 3923.648} C_VEL
LIN {X 0,Y 688.162,Z 780.81,A -85,B 0,C 180,E1 3928.912,E2 3928.912} C_VEL
LIN {X 0,Y 688.404,Z 780.81,A -85,B 0,C 180,E1 3934.154,E2 3934.154} C_VEL
LIN {X 0,Y 688.345,Z 780.81,A -85,B 0,C 180,E1 3939.442,E2 3939.442} C_VEL
LIN {X 0,Y 688.448,Z 780.81,A -85,B 0,C 180,E1 3944.733,E2 3944.733} C_VEL
LIN {X 0,Y 688.529,Z 780.81,A -85,B 0,C 180,E1 3949.892,E2 3949.892} C_VEL
LIN {X 0,Y 688.506,Z 780.81,A -85,B 0,C 180,E1 3954.966,E2 3954.966} C_VEL
LIN {X 0,Y 688.604,Z 780.81,A -85,B 0,C 180,E1 3960.002,E2 3960.002} C_VEL
LIN {X 0,Y 688.695,Z 780.81,A -85,B 0,C 180,E1 3965.036,E2 3965.036} C_VEL
LIN {X 0,Y 688.495,Z 780.81,A -85,B 0,C 180,E1 3970.113,E2 3970.113} C_VEL
LIN {X 0,Y 688.468,Z 780.81,A -85,B 0,C 180,E1 3975.27,E2 3975.27} C_VEL
LIN {X 0,Y 688.358,Z 780.81,A -85,B 0,C 180,E1 3980.561,E2 3980.561} C_VEL
LIN {X 0,Y 688.254,Z 780.81,A -85,B 0,C 180,E1 3986.045,E2 3986.045} C_VEL
LIN {X 0,Y 688.224,Z 780.81,A -85,B 0,C 180,E1 3991.097,E2 3991.097} C_VEL
LIN {X 0,Y 688.162,Z 780.81,A -85,B 0,C 180,E1 3996.357,E2 3996.357} C_VEL
LIN {X 0,Y 688.119,Z 780.81,A -85,B 0,C 180,E1 4001.701,E2 4001.701} C_VEL
LIN {X 0,Y 688.12,Z 780.81,A -85,B 0,C 180,E1 4006.434,E2 4006.434} C_VEL
LIN {X 0,Y 688.31,Z 780.81,A -85,B 0,C 180,E1 4012.208,E2 4012.208} C_VEL
LIN {X 0,Y 688.251,Z 780.818,A -85,B 0,C 180,E1 4014.278,E2 4014.278} C_VEL
LIN {X 0,Y 699.055,Z 805.854,A -85,B 0,C 180,E1 4015.171,E2 4015.171} C_VEL
LIN {X 0,Y 698.086,Z 851.406,A -85,B 0,C 180,E1 4016.116,E2 4016.116} C_VEL
LIN {X 0,Y 696.643,Z 894.007,A -85,B 0,C 180,E1 4017.504,E2 4017.504} C_VEL
LIN {X 0,Y 694.972,Z 936.769,A -85,B 0,C 180,E1 4019.465,E2 4019.465} C_VEL
LIN {X 0,Y 693.219,Z 977.481,A -85,B 0,C 180,E1 4021.964,E2 4021.964} C_VEL
LIN {X 0,Y 691.6,Z 1014.214,A -85,B 0,C 180,E1 4024.897,E2 4024.897} C_VEL
LIN {X 0,Y 690.363,Z 1045.871,A -85,B 0,C 180,E1 4028.155,E2 4028.155} C_VEL
LIN {X 0,Y 689.396,Z 1071.942,A -85,B 0,C 180,E1 4031.635,E2 4031.635} C_VEL
LIN {X 0,Y 689.041,Z 1089.853,A -85,B 0,C 180,E1 4034.755,E2 4034.755} C_VEL
LIN {X 0,Y 688.79,Z 1104.722,A -85,B 0,C 180,E1 4038.292,E2 4038.292} C_VEL
LIN {X 0,Y 688.703,Z 1114.262,A -85,B 0,C 180,E1 4041.801,E2 4041.801} C_VEL
LIN {X 0,Y 688.61,Z 1118.649,A -85,B 0,C 180,E1 4044.965,E2 4044.965} C_VEL
LIN {X 0,Y 688.6,Z 1118.811,A -85,B 0,C 180,E1 4048.743,E2 4048.743} C_VEL
LIN {X 0,Y 688.675,Z 1113.48,A -85,B 0,C 180,E1 4052.516,E2 4052.516} C_VEL
LIN {X 0,Y 688.776,Z 1103.406,A -85,B 0,C 180,E1 4055.982,E2 4055.982} C_VEL
LIN {X 0,Y 689.08,Z 1088.861,A -85,B 0,C 180,E1 4059.361,E2 4059.361} C_VEL
LIN {X 0,Y 689.723,Z 1066.777,A -85,B 0,C 180,E1 4063.04,E2 4063.04} C_VEL
LIN {X 0,Y 690.561,Z 1040.189,A -85,B 0,C 180,E1 4066.394,E2 4066.394} C_VEL
LIN {X 0,Y 691.742,Z 1009.881,A -85,B 0,C 180,E1 4069.392,E2 4069.392} C_VEL
LIN {X 0,Y 693.305,Z 975.302,A -85,B 0,C 180,E1 4072.095,E2 4072.095} C_VEL
LIN {X 0,Y 695.056,Z 934.719,A -85,B 0,C 180,E1 4074.555,E2 4074.555} C_VEL
LIN {X 0,Y 696.776,Z 889.887,A -85,B 0,C 180,E1 4076.571,E2 4076.571} C_VEL
LIN {X 0,Y 698.303,Z 842.671,A -85,B 0,C 180,E1 4078.024,E2 4078.024} C_VEL
LIN {X 0,Y 698.345,Z 803.563,A -85,B 0,C 180,E1 4078.807,E2 4078.807} C_VEL
LIN {X 0,Y 688.309,Z 780.81,A -85,B 0,C 180,E1 4079.651,E2 4079.651} C_VEL
LIN {X 0,Y 688.182,Z 780.81,A -85,B 0,C 180,E1 4084.814,E2 4084.814} C_VEL
LIN {X 0,Y 687.99,Z 780.81,A -85,B 0,C 180,E1 4089.768,E2 4089.768} C_VEL
LIN {X 0,Y 688.259,Z 780.81,A -85,B 0,C 180,E1 4094.635,E2 4094.635} C_VEL
LIN {X 0,Y 688.106,Z 780.81,A -85,B 0,C 180,E1 4100.448,E2 4100.448} C_VEL
LIN {X 0,Y 688.102,Z 780.81,A -85,B 0,C 180,E1 4105.186,E2 4105.186} C_VEL
LIN {X 0,Y 688.187,Z 780.81,A -85,B 0,C 180,E1 4109.67,E2 4109.67} C_VEL
LIN {X 0,Y 688.427,Z 780.81,A -85,B 0,C 180,E1 4114.154,E2 4114.154} C_VEL
LIN {X 0,Y 688.346,Z 780.81,A -85,B 0,C 180,E1 4119.438,E2 4119.438} C_VEL
LIN {X 0,Y 688.483,Z 780.81,A -85,B 0,C 180,E1 4124.73,E2 4124.73} C_VEL
LIN {X 0,Y 688.57,Z 780.81,A -85,B 0,C 180,E1 4129.888,E2 4129.888} C_VEL
LIN {X 0,Y 688.528,Z 780.81,A -85,B 0,C 180,E1 4134.963,E2 4134.963} C_VEL
LIN {X 0,Y 688.641,Z 780.81,A -85,B 0,C 180,E1 4139.998,E2 4139.998} C_VEL
LIN {X 0,Y 688.678,Z 780.81,A -85,B 0,C 180,E1 4145.032,E2 4145.032} C_VEL
LIN {X 0,Y 688.479,Z 780.81,A -85,B 0,C 180,E1 4150.109,E2 4150.109} C_VEL
LIN {X 0,Y 688.454,Z 780.81,A -85,B 0,C 180,E1 4155.267,E2 4155.267} C_VEL
LIN {X 0,Y 688.379,Z 780.81,A -85,B 0,C 180,E1 4160.056,E2 4160.056} C_VEL
LIN {X 0,Y 687.124,Z 780.81,A -85,B 0,C 180,E1 4160.775,E2 4160.775} C_VEL
LIN {X 0,Y 680.459,Z 780.81,A -85,B 0,C 180,E1 4162.729,E2 4162.729} C_VEL
LIN {X 0,Y 680.366,Z 780.81,A -85,B 0,C 180,E1 4162.914,E2 4162.914} C_VEL
LIN {X 0,Y 680.395,Z 780.81,A -85,B 0,C 180,E1 4167.793,E2 4167.793} C_VEL
LIN {X 0,Y 680.331,Z 780.81,A -85,B 0,C 180,E1 4172.431,E2 4172.431} C_VEL
LIN {X 0,Y 680.231,Z 780.81,A -85,B 0,C 180,E1 4176.895,E2 4176.895} C_VEL
LIN {X 0,Y 680.13,Z 780.81,A -85,B 0,C 180,E1 4181.789,E2 4181.789} C_VEL
LIN {X 0,Y 680.179,Z 780.81,A -85,B 0,C 180,E1 4187.137,E2 4187.137} C_VEL
LIN {X 0,Y 680.136,Z 780.81,A -85,B 0,C 180,E1 4191.53,E2 4191.53} C_VEL
LIN {X 0,Y 680.371,Z 780.81,A -85,B 0,C 180,E1 4196.382,E2 4196.382} C_VEL
LIN {X 0,Y 692.547,Z 808.991,A -85,B 0,C 180,E1 4197.408,E2 4197.408} C_VEL
LIN {X 0,Y 691.959,Z 865.934,A -85,B 0,C 180,E1 4198.219,E2 4198.219} C_VEL
LIN {X 0,Y 690.671,Z 910.519,A -85,B 0,C 180,E1 4199.386,E2 4199.386} C_VEL
LIN {X 0,Y 688.912,Z 952.186,A -85,B 0,C 180,E1 4200.99,E2 4200.99} C_VEL
